LIN {X 0,Y 298.924,Z 413.247,A -85,B 0,C 180,E1 -16471.347,E2 -16471.347} C_VEL
LIN {X 0,Y 298.607,Z 413.287,A -85,B 0,C 180,E1 -16475.401,E2 -16475.401} C_VEL
LIN {X 0,Y 298.427,Z 413.313,A -85,B 0,C 180,E1 -16478.123,E2 -16478.123} C_VEL
LIN {X 0,Y 298.154,Z 413.46,A -85,B 0,C 180,E1 -16479.497,E2 -16479.497} C_VEL
LIN {X 0,Y 297.871,Z 417.389,A -85,B 0,C 180,E1 -16483.646,E2 -16483.646} C_VEL
LIN {X 0,Y 297.437,Z 421.454,A -85,B 0,C 180,E1 -16487.888,E2 -16487.888} C_VEL
LIN {X 0,Y 297.33,Z 423.309,A -85,B 0,C 180,E1 -16489.768,E2 -16489.768} C_VEL
LIN {X 0,Y 300.977,Z 438.073,A -85,B 0,C 180,E1 -16490.771,E2 -16490.771} C_VEL
LIN {X 0,Y 303.389,Z 449.477,A -85,B 0,C 180,E1 -16491.754,E2 -16491.754} C_VEL
LIN {X 0,Y 304.98,Z 459.069,A -85,B 0,C 180,E1 -16492.741,E2 -16492.741} C_VEL
LIN {X 0,Y 303.705,Z 471.172,A -85,B 0,C 180,E1 -16494.07,E2 -16494.07} C_VEL
LIN {X 0,Y 302.343,Z 482.034,A -85,B 0,C 180,E1 -16495.588,E2 -16495.588} C_VEL
LIN {X 0,Y 300.988,Z 492.034,A -85,B 0,C 180,E1 -16497.325,E2 -16497.325} C_VEL
LIN {X 0,Y 299.841,Z 500.268,A -85,B 0,C 180,E1 -16499.101,E2 -16499.101} C_VEL
LIN {X 0,Y 298.694,Z 508.025,A -85,B 0,C 180,E1 -16501.173,E2 -16501.173} C_VEL
LIN {X 0,Y 298.042,Z 513.11,A -85,B 0,C 180,E1 -16502.843,E2 -16502.843} C_VEL
LIN {X 0,Y 297.488,Z 517.392,A -85,B 0,C 180,E1 -16504.539,E2 -16504.539} C_VEL
LIN {X 0,Y 296.854,Z 522.403,A -85,B 0,C 180,E1 -16507.174,E2 -16507.174} C_VEL
LIN {X 0,Y 296.651,Z 524.39,A -85,B 0,C 180,E1 -16508.574,E2 -16508.574} C_VEL
LIN {X 0,Y 296.39,Z 526.457,A -85,B 0,C 180,E1 -16510.643,E2 -16510.643} C_VEL
LIN {X 0,Y 296.318,Z 527.731,A -85,B 0,C 180,E1 -16513.456,E2 -16513.456} C_VEL
LIN {X 0,Y 296.377,Z 527.652,A -85,B 0,C 180,E1 -16515.347,E2 -16515.347} C_VEL
LIN {X 0,Y 296.62,Z 526.789,A -85,B 0,C 180,E1 -16517.264,E2 -16517.264} C_VEL
LIN {X 0,Y 297.047,Z 525.061,A -85,B 0,C 180,E1 -16519.208,E2 -16519.208} C_VEL
LIN {X 0,Y 297.66,Z 522.432,A -85,B 0,C 180,E1 -16521.182,E2 -16521.182} C_VEL
LIN {X 0,Y 298.415,Z 518.77,A -85,B 0,C 180,E1 -16523.199,E2 -16523.199} C_VEL
LIN {X 0,Y 299.433,Z 513.955,A -85,B 0,C 180,E1 -16525.232,E2 -16525.232} C_VEL
LIN {X 0,Y 300.922,Z 507.021,A -85,B 0,C 180,E1 -16527.509,E2 -16527.509} C_VEL
LIN {X 0,Y 302.361,Z 500.069,A -85,B 0,C 180,E1 -16529.317,E2 -16529.317} C_VEL
LIN {X 0,Y 304.36,Z 490.374,A -85,B 0,C 180,E1 -16531.336,E2 -16531.336} C_VEL
LIN {X 0,Y 306.05,Z 481.363,A -85,B 0,C 180,E1 -16532.849,E2 -16532.849} C_VEL
LIN {X 0,Y 307.84,Z 470.675,A -85,B 0,C 180,E1 -16534.293,E2 -16534.293} C_VEL
LIN {X 0,Y 308.746,Z 463.633,A -85,B 0,C 180,E1 -16535.095,E2 -16535.095} C_VEL
LIN {X 0,Y 307.123,Z 453.705,A -85,B 0,C 180,E1 -16536.322,E2 -16536.322} C_VEL
LIN {X 0,Y 304.252,Z 442.437,A -85,B 0,C 180,E1 -16537.597,E2 -16537.597} C_VEL
LIN {X 0,Y 300.037,Z 430.605,A -85,B 0,C 180,E1 -16538.846,E2 -16538.846} C_VEL
LIN {X 0,Y 298.096,Z 425.478,A -85,B 0,C 180,E1 -16539.333,E2 -16539.333} C_VEL
LIN {X 0,Y 298.371,Z 422.974,A -85,B 0,C 180,E1 -16542.169,E2 -16542.169} C_VEL
LIN {X 0,Y 298.739,Z 420.721,A -85,B 0,C 180,E1 -16545.002,E2 -16545.002} C_VEL
LIN {X 0,Y 298.89,Z 419.097,A -85,B 0,C 180,E1 -16547.183,E2 -16547.183} C_VEL
LIN {X 0,Y 298.349,Z 418.395,A -85,B 0,C 180,E1 -16548.301,E2 -16548.301} C_VEL
LIN {X 0,Y 295.711,Z 417.616,A -85,B 0,C 180,E1 -16550.135,E2 -16550.135} C_VEL
LIN {X 0,Y 292.496,Z 416.764,A -85,B 0,C 180,E1 -16552.386,E2 -16552.386} C_VEL
LIN {X 0,Y 292.069,Z 416.37,A -85,B 0,C 180,E1 -16553.16,E2 -16553.16} C_VEL
LIN {X 0,Y 291.789,Z 414.141,A -85,B 0,C 180,E1 -16557.239,E2 -16557.239} C_VEL
LIN {X 0,Y 291.977,Z 414.116,A -85,B 0,C 180,E1 -16560,E2 -16560} C_VEL
LIN {X 0,Y 291.786,Z 414.138,A -85,B 0,C 180,E1 -16562.761,E2 -16562.761} C_VEL
LIN {X 0,Y 291.743,Z 414.145,A -85,B 0,C 180,E1 -16566.918,E2 -16566.918} C_VEL
LIN {X 0,Y 291.626,Z 414.16,A -85,B 0,C 180,E1 -16569.712,E2 -16569.712} C_VEL
LIN {X 0,Y 291.518,Z 414.174,A -85,B 0,C 180,E1 -16573.951,E2 -16573.951} C_VEL
LIN {X 0,Y 291.483,Z 414.178,A -85,B 0,C 180,E1 -16576.818,E2 -16576.818} C_VEL
LIN {X 0,Y 291.447,Z 414.181,A -85,B 0,C 180,E1 -16579.875,E2 -16579.875} C_VEL
LIN {X 0,Y 291.397,Z 414.184,A -85,B 0,C 180,E1 -16584.206,E2 -16584.206} C_VEL
LIN {X 0,Y 291.42,Z 414.185,A -85,B 0,C 180,E1 -16587.272,E2 -16587.272} C_VEL
LIN {X 0,Y 291.335,Z 414.196,A -85,B 0,C 180,E1 -16590.437,E2 -16590.437} C_VEL
LIN {X 0,Y 291.342,Z 414.197,A -85,B 0,C 180,E1 -16593.699,E2 -16593.699} C_VEL
LIN {X 0,Y 291.384,Z 414.193,A -85,B 0,C 180,E1 -16595.371,E2 -16595.371} C_VEL
LIN {X 0,Y 291.576,Z 415.192,A -85,B 0,C 180,E1 -16597.307,E2 -16597.307} C_VEL
LIN {X 0,Y 291.962,Z 417.466,A -85,B 0,C 180,E1 -16600.537,E2 -16600.537} C_VEL
LIN {X 0,Y 292.454,Z 420.429,A -85,B 0,C 180,E1 -16604.179,E2 -16604.179} C_VEL
LIN {X 0,Y 293.009,Z 423.998,A -85,B 0,C 180,E1 -16608.035,E2 -16608.035} C_VEL
LIN {X 0,Y 293.495,Z 427.586,A -85,B 0,C 180,E1 -16611.495,E2 -16611.495} C_VEL
LIN {X 0,Y 293.526,Z 431.017,A -85,B 0,C 180,E1 -16614.496,E2 -16614.496} C_VEL
LIN {X 0,Y 292.934,Z 434.304,A -85,B 0,C 180,E1 -16617.11,E2 -16617.11} C_VEL
LIN {X 0,Y 291.919,Z 439.75,A -85,B 0,C 180,E1 -16621.217,E2 -16621.217} C_VEL
LIN {X 0,Y 291.619,Z 441.928,A -85,B 0,C 180,E1 -16622.82,E2 -16622.82} C_VEL
LIN {X 0,Y 292.601,Z 445.427,A -85,B 0,C 180,E1 -16623.121,E2 -16623.121} C_VEL
LIN {X 0,Y 296.153,Z 457.869,A -85,B 0,C 180,E1 -16624.282,E2 -16624.282} C_VEL
LIN {X 0,Y 298.394,Z 469.519,A -85,B 0,C 180,E1 -16625.468,E2 -16625.468} C_VEL
LIN {X 0,Y 299.71,Z 481.807,A -85,B 0,C 180,E1 -16626.864,E2 -16626.864} C_VEL
LIN {X 0,Y 299.877,Z 491.89,A -85,B 0,C 180,E1 -16628.159,E2 -16628.159} C_VEL
LIN {X 0,Y 298.451,Z 500.372,A -85,B 0,C 180,E1 -16629.316,E2 -16629.316} C_VEL
LIN {X 0,Y 296.409,Z 510.463,A -85,B 0,C 180,E1 -16630.973,E2 -16630.973} C_VEL
LIN {X 0,Y 294.65,Z 519.181,A -85,B 0,C 180,E1 -16632.756,E2 -16632.756} C_VEL
LIN {X 0,Y 293.172,Z 526.933,A -85,B 0,C 180,E1 -16634.711,E2 -16634.711} C_VEL
LIN {X 0,Y 291.663,Z 533.586,A -85,B 0,C 180,E1 -16636.767,E2 -16636.767} C_VEL
LIN {X 0,Y 290.708,Z 538.932,A -85,B 0,C 180,E1 -16638.849,E2 -16638.849} C_VEL
LIN {X 0,Y 290.033,Z 543.121,A -85,B 0,C 180,E1 -16640.938,E2 -16640.938} C_VEL
LIN {X 0,Y 289.609,Z 546.265,A -85,B 0,C 180,E1 -16643.031,E2 -16643.031} C_VEL
LIN {X 0,Y 289.475,Z 547.919,A -85,B 0,C 180,E1 -16644.513,E2 -16644.513} C_VEL
LIN {X 0,Y 289.475,Z 549.701,A -85,B 0,C 180,E1 -16647.217,E2 -16647.217} C_VEL
LIN {X 0,Y 289.459,Z 550.041,A -85,B 0,C 180,E1 -16648.609,E2 -16648.609} C_VEL
LIN {X 0,Y 289.498,Z 549.984,A -85,B 0,C 180,E1 -16650.001,E2 -16650.001} C_VEL
LIN {X 0,Y 289.467,Z 549.479,A -85,B 0,C 180,E1 -16651.392,E2 -16651.392} C_VEL
LIN {X 0,Y 289.49,Z 548.572,A -85,B 0,C 180,E1 -16652.784,E2 -16652.784} C_VEL
LIN {X 0,Y 289.467,Z 547.256,A -85,B 0,C 180,E1 -16654.177,E2 -16654.177} C_VEL
LIN {X 0,Y 289.555,Z 544.436,A -85,B 0,C 180,E1 -16656.271,E2 -16656.271} C_VEL
LIN {X 0,Y 289.846,Z 540.562,A -85,B 0,C 180,E1 -16658.366,E2 -16658.366} C_VEL
LIN {X 0,Y 290.351,Z 535.532,A -85,B 0,C 180,E1 -16660.46,E2 -16660.46} C_VEL
LIN {X 0,Y 291.089,Z 529.192,A -85,B 0,C 180,E1 -16662.551,E2 -16662.551} C_VEL
LIN {X 0,Y 292.231,Z 521.244,A -85,B 0,C 180,E1 -16664.627,E2 -16664.627} C_VEL
LIN {X 0,Y 293.404,Z 513.15,A -85,B 0,C 180,E1 -16666.347,E2 -16666.347} C_VEL
LIN {X 0,Y 294.728,Z 503.29,A -85,B 0,C 180,E1 -16668.059,E2 -16668.059} C_VEL
LIN {X 0,Y 296.272,Z 492.31,A -85,B 0,C 180,E1 -16669.577,E2 -16669.577} C_VEL
LIN {X 0,Y 296.655,Z 488.023,A -85,B 0,C 180,E1 -16670.092,E2 -16670.092} C_VEL
LIN {X 0,Y 295.753,Z 476.605,A -85,B 0,C 180,E1 -16671.347,E2 -16671.347} C_VEL
LIN {X 0,Y 294.197,Z 463.998,A -85,B 0,C 180,E1 -16672.472,E2 -16672.472} C_VEL
LIN {X 0,Y 292.088,Z 451.05,A -85,B 0,C 180,E1 -16673.378,E2 -16673.378} C_VEL
LIN {X 0,Y 290.748,Z 443.879,A -85,B 0,C 180,E1 -16673.794,E2 -16673.794} C_VEL
LIN {X 0,Y 291.476,Z 437.644,A -85,B 0,C 180,E1 -16678.046,E2 -16678.046} C_VEL
LIN {X 0,Y 292.238,Z 432.07,A -85,B 0,C 180,E1 -16681.943,E2 -16681.943} C_VEL
LIN {X 0,Y 292.974,Z 427.301,A -85,B 0,C 180,E1 -16685.352,E2 -16685.352} C_VEL
LIN {X 0,Y 292.931,Z 423.009,A -85,B 0,C 180,E1 -16688.594,E2 -16688.594} C_VEL
LIN {X 0,Y 292.132,Z 418.347,A -85,B 0,C 180,E1 -16692.347,E2 -16692.347} C_VEL
LIN {X 0,Y 291.364,Z 414.193,A -85,B 0,C 180,E1 -16696.046,E2 -16696.046} C_VEL
LIN {X 0,Y 291.38,Z 414.189,A -85,B 0,C 180,E1 -16700.519,E2 -16700.519} C_VEL
LIN {X 0,Y 291.406,Z 414.186,A -85,B 0,C 180,E1 -16702.919,E2 -16702.919} C_VEL
LIN {X 0,Y 291.346,Z 414.191,A -85,B 0,C 180,E1 -16706.302,E2 -16706.302} C_VEL
LIN {X 0,Y 291.389,Z 414.185,A -85,B 0,C 180,E1 -16710.26,E2 -16710.26} C_VEL
LIN {X 0,Y 291.414,Z 414.18,A -85,B 0,C 180,E1 -16714.271,E2 -16714.271} C_VEL
LIN {X 0,Y 291.383,Z 414.19,A -85,B 0,C 180,E1 -16717.299,E2 -16717.299} C_VEL
LIN {X 0,Y 291.459,Z 414.177,A -85,B 0,C 180,E1 -16720.27,E2 -16720.27} C_VEL
LIN {X 0,Y 291.557,Z 414.166,A -85,B 0,C 180,E1 -16724.624,E2 -16724.624} C_VEL
LIN {X 0,Y 291.538,Z 414.17,A -85,B 0,C 180,E1 -16728.881,E2 -16728.881} C_VEL
LIN {X 0,Y 291.71,Z 414.146,A -85,B 0,C 180,E1 -16731.688,E2 -16731.688} C_VEL
LIN {X 0,Y 291.631,Z 414.156,A -85,B 0,C 180,E1 -16734.468,E2 -16734.468} C_VEL
LIN {X 0,Y 291.889,Z 414.125,A -85,B 0,C 180,E1 -16738.62,E2 -16738.62} C_VEL
LIN {X 0,Y 291.89,Z 414.124,A -85,B 0,C 180,E1 -16741.38,E2 -16741.38} C_VEL
LIN {X 0,Y 291.747,Z 414.145,A -85,B 0,C 180,E1 -16746.918,E2 -16746.918} C_VEL
LIN {X 0,Y 291.631,Z 414.155,A -85,B 0,C 180,E1 -16749.712,E2 -16749.712} C_VEL
LIN {X 0,Y 291.523,Z 414.166,A -85,B 0,C 180,E1 -16753.95,E2 -16753.95} C_VEL
LIN {X 0,Y 291.488,Z 414.171,A -85,B 0,C 180,E1 -16756.818,E2 -16756.818} C_VEL
LIN {X 0,Y 291.452,Z 414.173,A -85,B 0,C 180,E1 -16759.875,E2 -16759.875} C_VEL
LIN {X 0,Y 291.402,Z 414.184,A -85,B 0,C 180,E1 -16764.205,E2 -16764.205} C_VEL
LIN {X 0,Y 291.427,Z 414.182,A -85,B 0,C 180,E1 -16767.271,E2 -16767.271} C_VEL
LIN {X 0,Y 291.338,Z 414.194,A -85,B 0,C 180,E1 -16770.437,E2 -16770.437} C_VEL
LIN {X 0,Y 291.346,Z 414.187,A -85,B 0,C 180,E1 -16773.698,E2 -16773.698} C_VEL
LIN {X 0,Y 291.377,Z 414.184,A -85,B 0,C 180,E1 -16777.254,E2 -16777.254} C_VEL
LIN {X 0,Y 291.334,Z 414.196,A -85,B 0,C 180,E1 -16780.642,E2 -16780.642} C_VEL
LIN {X 0,Y 291.291,Z 414.201,A -85,B 0,C 180,E1 -16784.402,E2 -16784.402} C_VEL
LIN {X 0,Y 291.328,Z 414.195,A -85,B 0,C 180,E1 -16788.404,E2 -16788.404} C_VEL
LIN {X 0,Y 291.366,Z 414.185,A -85,B 0,C 180,E1 -16791.16,E2 -16791.16} C_VEL
LIN {X 0,Y 291.387,Z 414.19,A -85,B 0,C 180,E1 -16794.629,E2 -16794.629} C_VEL
LIN {X 0,Y 291.372,Z 414.189,A -85,B 0,C 180,E1 -16797.95,E2 -16797.95} C_VEL
LIN {X 0,Y 291.378,Z 414.186,A -85,B 0,C 180,E1 -16801.158,E2 -16801.158} C_VEL
LIN {X 0,Y 291.414,Z 414.183,A -85,B 0,C 180,E1 -16804.271,E2 -16804.271} C_VEL
LIN {X 0,Y 291.391,Z 414.186,A -85,B 0,C 180,E1 -16807.3,E2 -16807.3} C_VEL
LIN {X 0,Y 291.46,Z 414.18,A -85,B 0,C 180,E1 -16810.27,E2 -16810.27} C_VEL
LIN {X 0,Y 291.557,Z 414.168,A -85,B 0,C 180,E1 -16814.623,E2 -16814.623} C_VEL
LIN {X 0,Y 291.539,Z 414.167,A -85,B 0,C 180,E1 -16818.88,E2 -16818.88} C_VEL
LIN {X 0,Y 291.712,Z 414.146,A -85,B 0,C 180,E1 -16821.688,E2 -16821.688} C_VEL
LIN {X 0,Y 291.632,Z 414.157,A -85,B 0,C 180,E1 -16824.468,E2 -16824.468} C_VEL
LIN {X 0,Y 291.89,Z 414.126,A -85,B 0,C 180,E1 -16828.62,E2 -16828.62} C_VEL
LIN {X 0,Y 291.89,Z 414.124,A -85,B 0,C 180,E1 -16831.379,E2 -16831.379} C_VEL
LIN {X 0,Y 291.568,Z 414.165,A -85,B 0,C 180,E1 -16835.532,E2 -16835.532} C_VEL
LIN {X 0,Y 291.318,Z 414.198,A -85,B 0,C 180,E1 -16838.46,E2 -16838.46} C_VEL
LIN {X 0,Y 291.074,Z 414.562,A -85,B 0,C 180,E1 -16839.73,E2 -16839.73} C_VEL
LIN {X 0,Y 290.787,Z 418.522,A -85,B 0,C 180,E1 -16843.986,E2 -16843.986} C_VEL
LIN {X 0,Y 290.341,Z 422.658,A -85,B 0,C 180,E1 -16848.341,E2 -16848.341} C_VEL
LIN {X 0,Y 290.311,Z 423.576,A -85,B 0,C 180,E1 -16849.299,E2 -16849.299} C_VEL
LIN {X 0,Y 293.844,Z 437.855,A -85,B 0,C 180,E1 -16850.291,E2 -16850.291} C_VEL
LIN {X 0,Y 296.457,Z 450.147,A -85,B 0,C 180,E1 -16851.375,E2 -16851.375} C_VEL
LIN {X 0,Y 298.112,Z 460.988,A -85,B 0,C 180,E1 -16852.525,E2 -16852.525} C_VEL
LIN {X 0,Y 296.663,Z 473.085,A -85,B 0,C 180,E1 -16853.934,E2 -16853.934} C_VEL
LIN {X 0,Y 295.246,Z 484.104,A -85,B 0,C 180,E1 -16855.559,E2 -16855.559} C_VEL
LIN {X 0,Y 293.834,Z 493.735,A -85,B 0,C 180,E1 -16857.342,E2 -16857.342} C_VEL
LIN {X 0,Y 292.58,Z 502.458,A -85,B 0,C 180,E1 -16859.347,E2 -16859.347} C_VEL
LIN {X 0,Y 291.586,Z 509.032,A -85,B 0,C 180,E1 -16861.211,E2 -16861.211} C_VEL
LIN {X 0,Y 290.871,Z 514.22,A -85,B 0,C 180,E1 -16863.012,E2 -16863.012} C_VEL
LIN {X 0,Y 290.115,Z 519.959,A -85,B 0,C 180,E1 -16865.548,E2 -16865.548} C_VEL
LIN {X 0,Y 289.613,Z 524.142,A -85,B 0,C 180,E1 -16868.169,E2 -16868.169} C_VEL
LIN {X 0,Y 289.292,Z 526.943,A -85,B 0,C 180,E1 -16870.989,E2 -16870.989} C_VEL
LIN {X 0,Y 289.227,Z 527.954,A -85,B 0,C 180,E1 -16873.199,E2 -16873.199} C_VEL
LIN {X 0,Y 289.272,Z 528.012,A -85,B 0,C 180,E1 -16875.205,E2 -16875.205} C_VEL
LIN {X 0,Y 289.51,Z 527.234,A -85,B 0,C 180,E1 -16877.179,E2 -16877.179} C_VEL
LIN {X 0,Y 289.932,Z 525.691,A -85,B 0,C 180,E1 -16879.119,E2 -16879.119} C_VEL
LIN {X 0,Y 290.531,Z 523.396,A -85,B 0,C 180,E1 -16881.028,E2 -16881.028} C_VEL
LIN {X 0,Y 291.202,Z 520.364,A -85,B 0,C 180,E1 -16882.889,E2 -16882.889} C_VEL
LIN {X 0,Y 292.379,Z 515.096,A -85,B 0,C 180,E1 -16885.295,E2 -16885.295} C_VEL
LIN {X 0,Y 293.919,Z 508.359,A -85,B 0,C 180,E1 -16887.643,E2 -16887.643} C_VEL
LIN {X 0,Y 295.487,Z 501.391,A -85,B 0,C 180,E1 -16889.563,E2 -16889.563} C_VEL
LIN {X 0,Y 297.407,Z 492.754,A -85,B 0,C 180,E1 -16891.468,E2 -16891.468} C_VEL
LIN {X 0,Y 299.46,Z 482.345,A -85,B 0,C 180,E1 -16893.305,E2 -16893.305} C_VEL
LIN {X 0,Y 301.37,Z 471.589,A -85,B 0,C 180,E1 -16894.813,E2 -16894.813} C_VEL
LIN {X 0,Y 302.242,Z 466.062,A -85,B 0,C 180,E1 -16895.459,E2 -16895.459} C_VEL
LIN {X 0,Y 301.069,Z 457.199,A -85,B 0,C 180,E1 -16896.619,E2 -16896.619} C_VEL
LIN {X 0,Y 298.662,Z 446.906,A -85,B 0,C 180,E1 -16897.883,E2 -16897.883} C_VEL
LIN {X 0,Y 294.909,Z 435.322,A -85,B 0,C 180,E1 -16899.193,E2 -16899.193} C_VEL
LIN {X 0,Y 291.251,Z 426.22,A -85,B 0,C 180,E1 -16900.173,E2 -16900.173} C_VEL
LIN {X 0,Y 291.162,Z 425.602,A -85,B 0,C 180,E1 -16900.249,E2 -16900.249} C_VEL
LIN {X 0,Y 291.656,Z 422.178,A -85,B 0,C 180,E1 -16904.629,E2 -16904.629} C_VEL
LIN {X 0,Y 291.921,Z 420.084,A -85,B 0,C 180,E1 -16907.486,E2 -16907.486} C_VEL
LIN {X 0,Y 292.135,Z 418.019,A -85,B 0,C 180,E1 -16910.517,E2 -16910.517} C_VEL
LIN {X 0,Y 292.069,Z 416.37,A -85,B 0,C 180,E1 -16913.16,E2 -16913.16} C_VEL
LIN {X 0,Y 291.228,Z 415.855,A -85,B 0,C 180,E1 -16914.304,E2 -16914.304} C_VEL
LIN {X 0,Y 288.277,Z 415.39,A -85,B 0,C 180,E1 -16916.174,E2 -16916.174} C_VEL
LIN {X 0,Y 285.901,Z 415.125,A -85,B 0,C 180,E1 -16917.695,E2 -16917.695} C_VEL
LIN {X 0,Y 284.93,Z 415.01,A -85,B 0,C 180,E1 -16918.873,E2 -16918.873} C_VEL
LIN {X 0,Y 284.871,Z 414.999,A -85,B 0,C 180,E1 -16919.272,E2 -16919.272} C_VEL
LIN {X 0,Y 284.741,Z 415.016,A -85,B 0,C 180,E1 -16922.83,E2 -16922.83} C_VEL
LIN {X 0,Y 284.695,Z 415.023,A -85,B 0,C 180,E1 -16927.09,E2 -16927.09} C_VEL
LIN {X 0,Y 284.563,Z 415.04,A -85,B 0,C 180,E1 -16929.956,E2 -16929.956} C_VEL
LIN {X 0,Y 284.478,Z 415.05,A -85,B 0,C 180,E1 -16934.303,E2 -16934.303} C_VEL
LIN {X 0,Y 284.422,Z 415.057,A -85,B 0,C 180,E1 -16937.249,E2 -16937.249} C_VEL
LIN {X 0,Y 284.375,Z 415.063,A -85,B 0,C 180,E1 -16940.243,E2 -16940.243} C_VEL
LIN {X 0,Y 284.366,Z 415.06,A -85,B 0,C 180,E1 -16943.876,E2 -16943.876} C_VEL
LIN {X 0,Y 284.394,Z 415.06,A -85,B 0,C 180,E1 -16947.174,E2 -16947.174} C_VEL
LIN {X 0,Y 284.293,Z 415.074,A -85,B 0,C 180,E1 -16951.275,E2 -16951.275} C_VEL
LIN {X 0,Y 284.343,Z 415.233,A -85,B 0,C 180,E1 -16954.645,E2 -16954.645} C_VEL
LIN {X 0,Y 284.716,Z 417.331,A -85,B 0,C 180,E1 -16958.105,E2 -16958.105} C_VEL
LIN {X 0,Y 285.185,Z 419.912,A -85,B 0,C 180,E1 -16961.712,E2 -16961.712} C_VEL
LIN {X 0,Y 285.665,Z 423.069,A -85,B 0,C 180,E1 -16965.518,E2 -16965.518} C_VEL
LIN {X 0,Y 286.294,Z 426.86,A -85,B 0,C 180,E1 -16969.552,E2 -16969.552} C_VEL
LIN {X 0,Y 286.584,Z 429.606,A -85,B 0,C 180,E1 -16972.188,E2 -16972.188} C_VEL
LIN {X 0,Y 286.553,Z 431.679,A -85,B 0,C 180,E1 -16974.034,E2 -16974.034} C_VEL
LIN {X 0,Y 285.833,Z 435.598,A -85,B 0,C 180,E1 -16977.254,E2 -16977.254} C_VEL
LIN {X 0,Y 284.724,Z 441.631,A -85,B 0,C 180,E1 -16981.907,E2 -16981.907} C_VEL
LIN {X 0,Y 285.569,Z 444.764,A -85,B 0,C 180,E1 -16982.169,E2 -16982.169} C_VEL
LIN {X 0,Y 288.858,Z 455.345,A -85,B 0,C 180,E1 -16983.231,E2 -16983.231} C_VEL
LIN {X 0,Y 291.371,Z 466.632,A -85,B 0,C 180,E1 -16984.421,E2 -16984.421} C_VEL
LIN {X 0,Y 292.858,Z 478.362,A -85,B 0,C 180,E1 -16985.773,E2 -16985.773} C_VEL
LIN {X 0,Y 293.353,Z 489.212,A -85,B 0,C 180,E1 -16987.184,E2 -16987.184} C_VEL
LIN {X 0,Y 293.064,Z 494.991,A -85,B 0,C 180,E1 -16987.995,E2 -16987.995} C_VEL
LIN {X 0,Y 290.931,Z 505.092,A -85,B 0,C 180,E1 -16989.497,E2 -16989.497} C_VEL
LIN {X 0,Y 288.953,Z 514.258,A -85,B 0,C 180,E1 -16991.2,E2 -16991.2} C_VEL
LIN {X 0,Y 287.079,Z 523.236,A -85,B 0,C 180,E1 -16993.283,E2 -16993.283} C_VEL
LIN {X 0,Y 285.534,Z 530.531,A -85,B 0,C 180,E1 -16995.388,E2 -16995.388} C_VEL
LIN {X 0,Y 284.305,Z 535.504,A -85,B 0,C 180,E1 -16997.146,E2 -16997.146} C_VEL
LIN {X 0,Y 283.449,Z 540.371,A -85,B 0,C 180,E1 -16999.284,E2 -16999.284} C_VEL
LIN {X 0,Y 282.807,Z 544.146,A -85,B 0,C 180,E1 -17001.426,E2 -17001.426} C_VEL
LIN {X 0,Y 282.556,Z 546.12,A -85,B 0,C 180,E1 -17002.857,E2 -17002.857} C_VEL
LIN {X 0,Y 282.371,Z 547.92,A -85,B 0,C 180,E1 -17004.608,E2 -17004.608} C_VEL
LIN {X 0,Y 282.379,Z 549.461,A -85,B 0,C 180,E1 -17007.147,E2 -17007.147} C_VEL
LIN {X 0,Y 282.38,Z 549.778,A -85,B 0,C 180,E1 -17008.574,E2 -17008.574} C_VEL
LIN {X 0,Y 282.415,Z 549.677,A -85,B 0,C 180,E1 -17010.001,E2 -17010.001} C_VEL
LIN {X 0,Y 282.388,Z 549.141,A -85,B 0,C 180,E1 -17011.427,E2 -17011.427} C_VEL
LIN {X 0,Y 282.417,Z 548.209,A -85,B 0,C 180,E1 -17012.853,E2 -17012.853} C_VEL
LIN {X 0,Y 282.409,Z 545.407,A -85,B 0,C 180,E1 -17015.474,E2 -17015.474} C_VEL
LIN {X 0,Y 282.672,Z 541.5,A -85,B 0,C 180,E1 -17017.86,E2 -17017.86} C_VEL
LIN {X 0,Y 283.128,Z 536.8,A -85,B 0,C 180,E1 -17020.007,E2 -17020.007} C_VEL
LIN {X 0,Y 283.944,Z 529.697,A -85,B 0,C 180,E1 -17022.508,E2 -17022.508} C_VEL
LIN {X 0,Y 285.128,Z 521.998,A -85,B 0,C 180,E1 -17024.635,E2 -17024.635} C_VEL
LIN {X 0,Y 286.385,Z 513.316,A -85,B 0,C 180,E1 -17026.554,E2 -17026.554} C_VEL
LIN {X 0,Y 287.774,Z 503.414,A -85,B 0,C 180,E1 -17028.327,E2 -17028.327} C_VEL
LIN {X 0,Y 289.357,Z 492.563,A -85,B 0,C 180,E1 -17029.88,E2 -17029.88} C_VEL
LIN {X 0,Y 289.697,Z 488.295,A -85,B 0,C 180,E1 -17030.41,E2 -17030.41} C_VEL
LIN {X 0,Y 288.705,Z 476.025,A -85,B 0,C 180,E1 -17031.797,E2 -17031.797} C_VEL
LIN {X 0,Y 287.077,Z 463.033,A -85,B 0,C 180,E1 -17032.983,E2 -17032.983} C_VEL
LIN {X 0,Y 284.861,Z 449.796,A -85,B 0,C 180,E1 -17033.92,E2 -17033.92} C_VEL
LIN {X 0,Y 283.728,Z 443.632,A -85,B 0,C 180,E1 -17034.283,E2 -17034.283} C_VEL
LIN {X 0,Y 284.56,Z 437.226,A -85,B 0,C 180,E1 -17038.791,E2 -17038.791} C_VEL
LIN {X 0,Y 285.403,Z 431.635,A -85,B 0,C 180,E1 -17042.803,E2 -17042.803} C_VEL
LIN {X 0,Y 285.979,Z 427.584,A -85,B 0,C 180,E1 -17045.807,E2 -17045.807} C_VEL
LIN {X 0,Y 285.853,Z 423.634,A -85,B 0,C 180,E1 -17048.872,E2 -17048.872} C_VEL
LIN {X 0,Y 285.143,Z 419.473,A -85,B 0,C 180,E1 -17052.318,E2 -17052.318} C_VEL
LIN {X 0,Y 284.306,Z 415.072,A -85,B 0,C 180,E1 -17056.199,E2 -17056.199} C_VEL
LIN {X 0,Y 284.308,Z 415.07,A -85,B 0,C 180,E1 -17060.024,E2 -17060.024} C_VEL
LIN {X 0,Y 284.332,Z 415.064,A -85,B 0,C 180,E1 -17063.614,E2 -17063.614} C_VEL
LIN {X 0,Y 284.309,Z 415.073,A -85,B 0,C 180,E1 -17067.19,E2 -17067.19} C_VEL
LIN {X 0,Y 284.36,Z 415.061,A -85,B 0,C 180,E1 -17070.376,E2 -17070.376} C_VEL
LIN {X 0,Y 284.376,Z 415.058,A -85,B 0,C 180,E1 -17073.586,E2 -17073.586} C_VEL
LIN {X 0,Y 284.368,Z 415.061,A -85,B 0,C 180,E1 -17076.707,E2 -17076.707} C_VEL
LIN {X 0,Y 284.405,Z 415.058,A -85,B 0,C 180,E1 -17081.262,E2 -17081.262} C_VEL
LIN {X 0,Y 284.494,Z 415.045,A -85,B 0,C 180,E1 -17084.459,E2 -17084.459} C_VEL
LIN {X 0,Y 284.49,Z 415.045,A -85,B 0,C 180,E1 -17088.601,E2 -17088.601} C_VEL
LIN {X 0,Y 284.66,Z 415.025,A -85,B 0,C 180,E1 -17091.481,E2 -17091.481} C_VEL
LIN {X 0,Y 284.602,Z 415.031,A -85,B 0,C 180,E1 -17094.331,E2 -17094.331} C_VEL
LIN {X 0,Y 284.855,Z 415,A -85,B 0,C 180,E1 -17098.586,E2 -17098.586} C_VEL
LIN {X 0,Y 284.856,Z 415,A -85,B 0,C 180,E1 -17101.414,E2 -17101.414} C_VEL
LIN {X 0,Y 284.699,Z 415.022,A -85,B 0,C 180,E1 -17107.09,E2 -17107.09} C_VEL
LIN {X 0,Y 284.568,Z 415.035,A -85,B 0,C 180,E1 -17109.955,E2 -17109.955} C_VEL
LIN {X 0,Y 284.483,Z 415.044,A -85,B 0,C 180,E1 -17114.303,E2 -17114.303} C_VEL
LIN {X 0,Y 284.427,Z 415.046,A -85,B 0,C 180,E1 -17117.248,E2 -17117.248} C_VEL
LIN {X 0,Y 284.38,Z 415.054,A -85,B 0,C 180,E1 -17120.242,E2 -17120.242} C_VEL
LIN {X 0,Y 284.37,Z 415.059,A -85,B 0,C 180,E1 -17123.875,E2 -17123.875} C_VEL
LIN {X 0,Y 284.401,Z 415.058,A -85,B 0,C 180,E1 -17127.174,E2 -17127.174} C_VEL
LIN {X 0,Y 284.297,Z 415.068,A -85,B 0,C 180,E1 -17131.274,E2 -17131.274} C_VEL
LIN {X 0,Y 284.342,Z 415.056,A -85,B 0,C 180,E1 -17135.348,E2 -17135.348} C_VEL
LIN {X 0,Y 284.313,Z 415.064,A -85,B 0,C 180,E1 -17138.169,E2 -17138.169} C_VEL
LIN {X 0,Y 284.27,Z 415.073,A -85,B 0,C 180,E1 -17142.124,E2 -17142.124} C_VEL
LIN {X 0,Y 284.256,Z 415.075,A -85,B 0,C 180,E1 -17146.189,E2 -17146.189} C_VEL
LIN {X 0,Y 284.308,Z 415.065,A -85,B 0,C 180,E1 -17150.024,E2 -17150.024} C_VEL
LIN {X 0,Y 284.352,Z 415.06,A -85,B 0,C 180,E1 -17153.617,E2 -17153.617} C_VEL
LIN {X 0,Y 284.309,Z 415.068,A -85,B 0,C 180,E1 -17157.189,E2 -17157.189} C_VEL
LIN {X 0,Y 284.357,Z 415.065,A -85,B 0,C 180,E1 -17160.375,E2 -17160.375} C_VEL
LIN {X 0,Y 284.376,Z 415.056,A -85,B 0,C 180,E1 -17163.586,E2 -17163.586} C_VEL
LIN {X 0,Y 284.371,Z 415.063,A -85,B 0,C 180,E1 -17166.707,E2 -17166.707} C_VEL
LIN {X 0,Y 284.405,Z 415.054,A -85,B 0,C 180,E1 -17171.261,E2 -17171.261} C_VEL
LIN {X 0,Y 284.494,Z 415.05,A -85,B 0,C 180,E1 -17174.459,E2 -17174.459} C_VEL
LIN {X 0,Y 284.49,Z 415.047,A -85,B 0,C 180,E1 -17178.601,E2 -17178.601} C_VEL
LIN {X 0,Y 284.662,Z 415.024,A -85,B 0,C 180,E1 -17181.481,E2 -17181.481} C_VEL
LIN {X 0,Y 284.603,Z 415.033,A -85,B 0,C 180,E1 -17184.331,E2 -17184.331} C_VEL
LIN {X 0,Y 284.856,Z 415.003,A -85,B 0,C 180,E1 -17188.586,E2 -17188.586} C_VEL
LIN {X 0,Y 284.856,Z 415,A -85,B 0,C 180,E1 -17191.413,E2 -17191.413} C_VEL
LIN {X 0,Y 284.528,Z 415.042,A -85,B 0,C 180,E1 -17195.67,E2 -17195.67} C_VEL
LIN {X 0,Y 284.265,Z 415.076,A -85,B 0,C 180,E1 -17198.53,E2 -17198.53} C_VEL
LIN {X 0,Y 284.048,Z 415.357,A -85,B 0,C 180,E1 -17199.613,E2 -17199.613} C_VEL
LIN {X 0,Y 283.771,Z 418.293,A -85,B 0,C 180,E1 -17202.879,E2 -17202.879} C_VEL
LIN {X 0,Y 283.493,Z 421.046,A -85,B 0,C 180,E1 -17205.824,E2 -17205.824} C_VEL
LIN {X 0,Y 283.282,Z 423.967,A -85,B 0,C 180,E1 -17208.815,E2 -17208.815} C_VEL
LIN {X 0,Y 286.608,Z 437.123,A -85,B 0,C 180,E1 -17209.746,E2 -17209.746} C_VEL
LIN {X 0,Y 289.204,Z 449.093,A -85,B 0,C 180,E1 -17210.818,E2 -17210.818} C_VEL
LIN {X 0,Y 291.146,Z 460.447,A -85,B 0,C 180,E1 -17212.045,E2 -17212.045} C_VEL
LIN {X 0,Y 290.64,Z 466.848,A -85,B 0,C 180,E1 -17212.761,E2 -17212.761} C_VEL
LIN {X 0,Y 289.262,Z 477.904,A -85,B 0,C 180,E1 -17214.227,E2 -17214.227} C_VEL
LIN {X 0,Y 287.908,Z 487.208,A -85,B 0,C 180,E1 -17215.744,E2 -17215.744} C_VEL
LIN {X 0,Y 286.704,Z 495.369,A -85,B 0,C 180,E1 -17217.362,E2 -17217.362} C_VEL
LIN {X 0,Y 285.355,Z 504.186,A -85,B 0,C 180,E1 -17219.509,E2 -17219.509} C_VEL
LIN {X 0,Y 284.348,Z 511.022,A -85,B 0,C 180,E1 -17221.605,E2 -17221.605} C_VEL
LIN {X 0,Y 283.474,Z 516.972,A -85,B 0,C 180,E1 -17223.905,E2 -17223.905} C_VEL
LIN {X 0,Y 282.996,Z 520.734,A -85,B 0,C 180,E1 -17225.756,E2 -17225.756} C_VEL
LIN {X 0,Y 282.479,Z 524.808,A -85,B 0,C 180,E1 -17228.461,E2 -17228.461} C_VEL
LIN {X 0,Y 282.244,Z 526.685,A -85,B 0,C 180,E1 -17230.346,E2 -17230.346} C_VEL
LIN {X 0,Y 282.139,Z 527.883,A -85,B 0,C 180,E1 -17232.264,E2 -17232.264} C_VEL
LIN {X 0,Y 282.126,Z 528.367,A -85,B 0,C 180,E1 -17234.226,E2 -17234.226} C_VEL
LIN {X 0,Y 282.283,Z 528.051,A -85,B 0,C 180,E1 -17236.22,E2 -17236.22} C_VEL
LIN {X 0,Y 282.633,Z 526.95,A -85,B 0,C 180,E1 -17238.243,E2 -17238.243} C_VEL
LIN {X 0,Y 283.174,Z 525.004,A -85,B 0,C 180,E1 -17240.297,E2 -17240.297} C_VEL
LIN {X 0,Y 284.176,Z 521.06,A -85,B 0,C 180,E1 -17243.011,E2 -17243.011} C_VEL
LIN {X 0,Y 285.428,Z 515.915,A -85,B 0,C 180,E1 -17245.506,E2 -17245.506} C_VEL
LIN {X 0,Y 286.908,Z 509.821,A -85,B 0,C 180,E1 -17247.741,E2 -17247.741} C_VEL
LIN {X 0,Y 288.439,Z 503.393,A -85,B 0,C 180,E1 -17249.63,E2 -17249.63} C_VEL
LIN {X 0,Y 290.464,Z 494.843,A -85,B 0,C 180,E1 -17251.651,E2 -17251.651} C_VEL
LIN {X 0,Y 292.341,Z 486.212,A -85,B 0,C 180,E1 -17253.302,E2 -17253.302} C_VEL
LIN {X 0,Y 294.276,Z 476.252,A -85,B 0,C 180,E1 -17254.853,E2 -17254.853} C_VEL
LIN {X 0,Y 295.801,Z 467.169,A -85,B 0,C 180,E1 -17256.013,E2 -17256.013} C_VEL
LIN {X 0,Y 294.466,Z 457.672,A -85,B 0,C 180,E1 -17257.324,E2 -17257.324} C_VEL
LIN {X 0,Y 291.968,Z 447.356,A -85,B 0,C 180,E1 -17258.649,E2 -17258.649} C_VEL
LIN {X 0,Y 287.89,Z 435.363,A -85,B 0,C 180,E1 -17260.104,E2 -17260.104} C_VEL
LIN {X 0,Y 285.055,Z 428.698,A -85,B 0,C 180,E1 -17260.893,E2 -17260.893} C_VEL
LIN {X 0,Y 284.223,Z 425.951,A -85,B 0,C 180,E1 -17261.186,E2 -17261.186} C_VEL
LIN {X 0,Y 284.741,Z 422.568,A -85,B 0,C 180,E1 -17265.711,E2 -17265.711} C_VEL
LIN {X 0,Y 284.995,Z 420.554,A -85,B 0,C 180,E1 -17268.622,E2 -17268.622} C_VEL
LIN {X 0,Y 285.183,Z 418.685,A -85,B 0,C 180,E1 -17271.497,E2 -17271.497} C_VEL
LIN {X 0,Y 284.932,Z 417.06,A -85,B 0,C 180,E1 -17274.338,E2 -17274.338} C_VEL
LIN {X 0,Y 284.854,Z 415.004,A -85,B 0,C 180,E1 -17278.586,E2 -17278.586} C_VEL
LIN {X 0,Y 284.871,Z 414.999,A -85,B 0,C 180,E1 -17279.272,E2 -17279.272} C_VEL
LIN {X 0,Y 284.201,Z 415.084,A -85,B 0,C 180,E1 -17280.451,E2 -17280.451} C_VEL
LIN {X 0,Y 281.167,Z 415.46,A -85,B 0,C 180,E1 -17282.365,E2 -17282.365} C_VEL
LIN {X 0,Y 278.612,Z 415.781,A -85,B 0,C 180,E1 -17283.922,E2 -17283.922} C_VEL
LIN {X 0,Y 277.582,Z 415.91,A -85,B 0,C 180,E1 -17285.133,E2 -17285.133} C_VEL
LIN {X 0,Y 277.535,Z 415.914,A -85,B 0,C 180,E1 -17285.543,E2 -17285.543} C_VEL
LIN {X 0,Y 277.612,Z 415.906,A -85,B 0,C 180,E1 -17288.737,E2 -17288.737} C_VEL
LIN {X 0,Y 277.413,Z 415.93,A -85,B 0,C 180,E1 -17293.18,E2 -17293.18} C_VEL
LIN {X 0,Y 277.403,Z 415.931,A -85,B 0,C 180,E1 -17296.182,E2 -17296.182} C_VEL
LIN {X 0,Y 277.342,Z 415.939,A -85,B 0,C 180,E1 -17300.35,E2 -17300.35} C_VEL
LIN {X 0,Y 277.316,Z 415.937,A -85,B 0,C 180,E1 -17304.171,E2 -17304.171} C_VEL
LIN {X 0,Y 277.323,Z 415.942,A -85,B 0,C 180,E1 -17307.506,E2 -17307.506} C_VEL
LIN {X 0,Y 277.269,Z 415.948,A -85,B 0,C 180,E1 -17310.482,E2 -17310.482} C_VEL
LIN {X 0,Y 277.287,Z 416.154,A -85,B 0,C 180,E1 -17313.239,E2 -17313.239} C_VEL
LIN {X 0,Y 277.572,Z 417.557,A -85,B 0,C 180,E1 -17315.884,E2 -17315.884} C_VEL
LIN {X 0,Y 277.919,Z 419.664,A -85,B 0,C 180,E1 -17319.213,E2 -17319.213} C_VEL
LIN {X 0,Y 278.406,Z 422.406,A -85,B 0,C 180,E1 -17322.968,E2 -17322.968} C_VEL
LIN {X 0,Y 278.966,Z 425.936,A -85,B 0,C 180,E1 -17327.141,E2 -17327.141} C_VEL
LIN {X 0,Y 279.263,Z 427.793,A -85,B 0,C 180,E1 -17329.133,E2 -17329.133} C_VEL
LIN {X 0,Y 279.49,Z 429.864,A -85,B 0,C 180,E1 -17331.217,E2 -17331.217} C_VEL
LIN {X 0,Y 279.559,Z 432.373,A -85,B 0,C 180,E1 -17333.559,E2 -17333.559} C_VEL
LIN {X 0,Y 279.037,Z 435.603,A -85,B 0,C 180,E1 -17336.352,E2 -17336.352} C_VEL
LIN {X 0,Y 277.886,Z 441.268,A -85,B 0,C 180,E1 -17340.905,E2 -17340.905} C_VEL
LIN {X 0,Y 279,Z 444.991,A -85,B 0,C 180,E1 -17341.265,E2 -17341.265} C_VEL
LIN {X 0,Y 282.489,Z 456.404,A -85,B 0,C 180,E1 -17342.478,E2 -17342.478} C_VEL
LIN {X 0,Y 284.965,Z 467.644,A -85,B 0,C 180,E1 -17343.755,E2 -17343.755} C_VEL
LIN {X 0,Y 286.423,Z 479.622,A -85,B 0,C 180,E1 -17345.214,E2 -17345.214} C_VEL
LIN {X 0,Y 286.831,Z 490.082,A -85,B 0,C 180,E1 -17346.641,E2 -17346.641} C_VEL
LIN {X 0,Y 286.289,Z 496.878,A -85,B 0,C 180,E1 -17347.636,E2 -17347.636} C_VEL
LIN {X 0,Y 283.885,Z 507.474,A -85,B 0,C 180,E1 -17349.343,E2 -17349.343} C_VEL
LIN {X 0,Y 281.864,Z 516.167,A -85,B 0,C 180,E1 -17351.087,E2 -17351.087} C_VEL
LIN {X 0,Y 280.032,Z 524.736,A -85,B 0,C 180,E1 -17353.226,E2 -17353.226} C_VEL
LIN {X 0,Y 278.372,Z 531.664,A -85,B 0,C 180,E1 -17355.377,E2 -17355.377} C_VEL
LIN {X 0,Y 277.009,Z 537.258,A -85,B 0,C 180,E1 -17357.547,E2 -17357.547} C_VEL
LIN {X 0,Y 276.192,Z 541.685,A -85,B 0,C 180,E1 -17359.74,E2 -17359.74} C_VEL
LIN {X 0,Y 275.772,Z 544.048,A -85,B 0,C 180,E1 -17361.205,E2 -17361.205} C_VEL
LIN {X 0,Y 275.492,Z 545.986,A -85,B 0,C 180,E1 -17362.672,E2 -17362.672} C_VEL
LIN {X 0,Y 275.25,Z 548.535,A -85,B 0,C 180,E1 -17365.607,E2 -17365.607} C_VEL
LIN {X 0,Y 275.286,Z 549.221,A -85,B 0,C 180,E1 -17367.074,E2 -17367.074} C_VEL
LIN {X 0,Y 275.303,Z 549.513,A -85,B 0,C 180,E1 -17368.538,E2 -17368.538} C_VEL
LIN {X 0,Y 275.334,Z 549.364,A -85,B 0,C 180,E1 -17370.001,E2 -17370.001} C_VEL
LIN {X 0,Y 275.311,Z 548.804,A -85,B 0,C 180,E1 -17371.463,E2 -17371.463} C_VEL
LIN {X 0,Y 275.321,Z 547.846,A -85,B 0,C 180,E1 -17372.927,E2 -17372.927} C_VEL
LIN {X 0,Y 275.326,Z 545.227,A -85,B 0,C 180,E1 -17375.423,E2 -17375.423} C_VEL
LIN {X 0,Y 275.601,Z 540.997,A -85,B 0,C 180,E1 -17378.063,E2 -17378.063} C_VEL
LIN {X 0,Y 276.111,Z 536.236,A -85,B 0,C 180,E1 -17380.264,E2 -17380.264} C_VEL
LIN {X 0,Y 276.979,Z 529.064,A -85,B 0,C 180,E1 -17382.828,E2 -17382.828} C_VEL
LIN {X 0,Y 278.183,Z 521.243,A -85,B 0,C 180,E1 -17385.009,E2 -17385.009} C_VEL
LIN {X 0,Y 279.315,Z 514.077,A -85,B 0,C 180,E1 -17386.647,E2 -17386.647} C_VEL
LIN {X 0,Y 280.826,Z 503.52,A -85,B 0,C 180,E1 -17388.608,E2 -17388.608} C_VEL
LIN {X 0,Y 282.452,Z 492.774,A -85,B 0,C 180,E1 -17390.197,E2 -17390.197} C_VEL
LIN {X 0,Y 282.724,Z 488.514,A -85,B 0,C 180,E1 -17390.747,E2 -17390.747} C_VEL
LIN {X 0,Y 281.907,Z 477.62,A -85,B 0,C 180,E1 -17392.044,E2 -17392.044} C_VEL
LIN {X 0,Y 280.396,Z 464.931,A -85,B 0,C 180,E1 -17393.273,E2 -17393.273} C_VEL
LIN {X 0,Y 278.293,Z 451.753,A -85,B 0,C 180,E1 -17394.284,E2 -17394.284} C_VEL
LIN {X 0,Y 276.744,Z 443.37,A -85,B 0,C 180,E1 -17394.812,E2 -17394.812} C_VEL
LIN {X 0,Y 277.635,Z 436.785,A -85,B 0,C 180,E1 -17399.579,E2 -17399.579} C_VEL
LIN {X 0,Y 278.527,Z 431.209,A -85,B 0,C 180,E1 -17403.719,E2 -17403.719} C_VEL
LIN {X 0,Y 278.943,Z 427.873,A -85,B 0,C 180,E1 -17406.269,E2 -17406.269} C_VEL
LIN {X 0,Y 278.782,Z 424.388,A -85,B 0,C 180,E1 -17409.068,E2 -17409.068} C_VEL
LIN {X 0,Y 277.979,Z 419.947,A -85,B 0,C 180,E1 -17412.845,E2 -17412.845} C_VEL
LIN {X 0,Y 277.249,Z 415.951,A -85,B 0,C 180,E1 -17416.56,E2 -17416.56} C_VEL
LIN {X 0,Y 277.235,Z 415.953,A -85,B 0,C 180,E1 -17420.672,E2 -17420.672} C_VEL
LIN {X 0,Y 277.285,Z 415.939,A -85,B 0,C 180,E1 -17424.341,E2 -17424.341} C_VEL
LIN {X 0,Y 277.246,Z 415.949,A -85,B 0,C 180,E1 -17427.836,E2 -17427.836} C_VEL
LIN {X 0,Y 277.29,Z 415.943,A -85,B 0,C 180,E1 -17431.212,E2 -17431.212} C_VEL
LIN {X 0,Y 277.313,Z 415.937,A -85,B 0,C 180,E1 -17434.479,E2 -17434.479} C_VEL
LIN {X 0,Y 277.287,Z 415.944,A -85,B 0,C 180,E1 -17437.655,E2 -17437.655} C_VEL
LIN {X 0,Y 277.347,Z 415.937,A -85,B 0,C 180,E1 -17440.766,E2 -17440.766} C_VEL
LIN {X 0,Y 277.436,Z 415.926,A -85,B 0,C 180,E1 -17445.326,E2 -17445.326} C_VEL
LIN {X 0,Y 277.508,Z 415.914,A -85,B 0,C 180,E1 -17449.789,E2 -17449.789} C_VEL
LIN {X 0,Y 277.654,Z 415.899,A -85,B 0,C 180,E1 -17452.729,E2 -17452.729} C_VEL
LIN {X 0,Y 277.821,Z 415.876,A -85,B 0,C 180,E1 -17458.55,E2 -17458.55} C_VEL
LIN {X 0,Y 277.822,Z 415.876,A -85,B 0,C 180,E1 -17461.449,E2 -17461.449} C_VEL
LIN {X 0,Y 277.654,Z 415.898,A -85,B 0,C 180,E1 -17467.271,E2 -17467.271} C_VEL
LIN {X 0,Y 277.508,Z 415.915,A -85,B 0,C 180,E1 -17470.211,E2 -17470.211} C_VEL
LIN {X 0,Y 277.436,Z 415.924,A -85,B 0,C 180,E1 -17474.674,E2 -17474.674} C_VEL
LIN {X 0,Y 277.346,Z 415.93,A -85,B 0,C 180,E1 -17479.234,E2 -17479.234} C_VEL
LIN {X 0,Y 277.321,Z 415.937,A -85,B 0,C 180,E1 -17484.17,E2 -17484.17} C_VEL
LIN {X 0,Y 277.329,Z 415.937,A -85,B 0,C 180,E1 -17487.506,E2 -17487.506} C_VEL
LIN {X 0,Y 277.273,Z 415.946,A -85,B 0,C 180,E1 -17490.481,E2 -17490.481} C_VEL
LIN {X 0,Y 277.248,Z 415.942,A -85,B 0,C 180,E1 -17493.896,E2 -17493.896} C_VEL
LIN {X 0,Y 277.269,Z 415.939,A -85,B 0,C 180,E1 -17497.469,E2 -17497.469} C_VEL
LIN {X 0,Y 277.21,Z 415.952,A -85,B 0,C 180,E1 -17501.236,E2 -17501.236} C_VEL
LIN {X 0,Y 277.202,Z 415.953,A -85,B 0,C 180,E1 -17505.226,E2 -17505.226} C_VEL
LIN {X 0,Y 277.224,Z 415.946,A -85,B 0,C 180,E1 -17509.512,E2 -17509.512} C_VEL
LIN {X 0,Y 277.283,Z 415.942,A -85,B 0,C 180,E1 -17512.533,E2 -17512.533} C_VEL
LIN {X 0,Y 277.256,Z 415.947,A -85,B 0,C 180,E1 -17516.105,E2 -17516.105} C_VEL
LIN {X 0,Y 277.263,Z 415.945,A -85,B 0,C 180,E1 -17519.538,E2 -17519.538} C_VEL
LIN {X 0,Y 277.357,Z 415.932,A -85,B 0,C 180,E1 -17522.864,E2 -17522.864} C_VEL
LIN {X 0,Y 277.33,Z 415.938,A -85,B 0,C 180,E1 -17526.079,E2 -17526.079} C_VEL
LIN {X 0,Y 277.347,Z 415.935,A -85,B 0,C 180,E1 -17530.766,E2 -17530.766} C_VEL
LIN {X 0,Y 277.437,Z 415.924,A -85,B 0,C 180,E1 -17535.326,E2 -17535.326} C_VEL
LIN {X 0,Y 277.509,Z 415.915,A -85,B 0,C 180,E1 -17539.788,E2 -17539.788} C_VEL
LIN {X 0,Y 277.656,Z 415.898,A -85,B 0,C 180,E1 -17542.729,E2 -17542.729} C_VEL
LIN {X 0,Y 277.822,Z 415.88,A -85,B 0,C 180,E1 -17548.55,E2 -17548.55} C_VEL
LIN {X 0,Y 277.822,Z 415.876,A -85,B 0,C 180,E1 -17551.449,E2 -17551.449} C_VEL
LIN {X 0,Y 277.488,Z 415.92,A -85,B 0,C 180,E1 -17555.814,E2 -17555.814} C_VEL
LIN {X 0,Y 277.175,Z 415.959,A -85,B 0,C 180,E1 -17558.75,E2 -17558.75} C_VEL
LIN {X 0,Y 277.02,Z 416.139,A -85,B 0,C 180,E1 -17559.491,E2 -17559.491} C_VEL
LIN {X 0,Y 276.68,Z 419.458,A -85,B 0,C 180,E1 -17563.215,E2 -17563.215} C_VEL
LIN {X 0,Y 276.367,Z 422.191,A -85,B 0,C 180,E1 -17566.243,E2 -17566.243} C_VEL
LIN {X 0,Y 276.259,Z 424.141,A -85,B 0,C 180,E1 -17568.301,E2 -17568.301} C_VEL
LIN {X 0,Y 279.671,Z 437.593,A -85,B 0,C 180,E1 -17569.278,E2 -17569.278} C_VEL
LIN {X 0,Y 282.295,Z 449.696,A -85,B 0,C 180,E1 -17570.397,E2 -17570.397} C_VEL
LIN {X 0,Y 284.348,Z 461.804,A -85,B 0,C 180,E1 -17571.761,E2 -17571.761} C_VEL
LIN {X 0,Y 282.968,Z 473.709,A -85,B 0,C 180,E1 -17573.225,E2 -17573.225} C_VEL
LIN {X 0,Y 281.434,Z 484.695,A -85,B 0,C 180,E1 -17574.922,E2 -17574.922} C_VEL
LIN {X 0,Y 279.879,Z 494.681,A -85,B 0,C 180,E1 -17576.871,E2 -17576.871} C_VEL
LIN {X 0,Y 278.501,Z 503.671,A -85,B 0,C 180,E1 -17579.062,E2 -17579.062} C_VEL
LIN {X 0,Y 277.337,Z 511.067,A -85,B 0,C 180,E1 -17581.348,E2 -17581.348} C_VEL
LIN {X 0,Y 276.506,Z 516.556,A -85,B 0,C 180,E1 -17583.48,E2 -17583.48} C_VEL
LIN {X 0,Y 275.874,Z 521.329,A -85,B 0,C 180,E1 -17585.868,E2 -17585.868} C_VEL
LIN {X 0,Y 275.328,Z 525.378,A -85,B 0,C 180,E1 -17588.709,E2 -17588.709} C_VEL
LIN {X 0,Y 275.167,Z 526.637,A -85,B 0,C 180,E1 -17589.984,E2 -17589.984} C_VEL
LIN {X 0,Y 275.044,Z 528.098,A -85,B 0,C 180,E1 -17592.182,E2 -17592.182} C_VEL
LIN {X 0,Y 275.033,Z 528.641,A -85,B 0,C 180,E1 -17594.316,E2 -17594.316} C_VEL
LIN {X 0,Y 275.231,Z 528.336,A -85,B 0,C 180,E1 -17596.414,E2 -17596.414} C_VEL
LIN {X 0,Y 275.585,Z 527.261,A -85,B 0,C 180,E1 -17598.467,E2 -17598.467} C_VEL
LIN {X 0,Y 276.138,Z 525.439,A -85,B 0,C 180,E1 -17600.485,E2 -17600.485} C_VEL
LIN {X 0,Y 277.227,Z 521.419,A -85,B 0,C 180,E1 -17603.351,E2 -17603.351} C_VEL
LIN {X 0,Y 278.54,Z 516.438,A -85,B 0,C 180,E1 -17605.848,E2 -17605.848} C_VEL
LIN {X 0,Y 280.152,Z 510.178,A -85,B 0,C 180,E1 -17608.21,E2 -17608.21} C_VEL
LIN {X 0,Y 282.034,Z 502.756,A -85,B 0,C 180,E1 -17610.416,E2 -17610.416} C_VEL
LIN {X 0,Y 284.148,Z 494.346,A -85,B 0,C 180,E1 -17612.409,E2 -17612.409} C_VEL
LIN {X 0,Y 286.088,Z 485.793,A -85,B 0,C 180,E1 -17614.052,E2 -17614.052} C_VEL
LIN {X 0,Y 288.209,Z 475.15,A -85,B 0,C 180,E1 -17615.701,E2 -17615.701} C_VEL
LIN {X 0,Y 289.361,Z 468.527,A -85,B 0,C 180,E1 -17616.565,E2 -17616.565} C_VEL
LIN {X 0,Y 287.914,Z 458.394,A -85,B 0,C 180,E1 -17618.031,E2 -17618.031} C_VEL
LIN {X 0,Y 285.256,Z 447.533,A -85,B 0,C 180,E1 -17619.505,E2 -17619.505} C_VEL
LIN {X 0,Y 281.254,Z 436.129,A -85,B 0,C 180,E1 -17620.979,E2 -17620.979} C_VEL
LIN {X 0,Y 278.312,Z 429.392,A -85,B 0,C 180,E1 -17621.838,E2 -17621.838} C_VEL
LIN {X 0,Y 277.304,Z 426.312,A -85,B 0,C 180,E1 -17622.199,E2 -17622.199} C_VEL
LIN {X 0,Y 277.679,Z 424.032,A -85,B 0,C 180,E1 -17625.339,E2 -17625.339} C_VEL
LIN {X 0,Y 277.99,Z 422.005,A -85,B 0,C 180,E1 -17628.331,E2 -17628.331} C_VEL
LIN {X 0,Y 278.197,Z 420.136,A -85,B 0,C 180,E1 -17631.282,E2 -17631.282} C_VEL
LIN {X 0,Y 277.983,Z 418.513,A -85,B 0,C 180,E1 -17634.196,E2 -17634.196} C_VEL
LIN {X 0,Y 277.879,Z 416.336,A -85,B 0,C 180,E1 -17638.551,E2 -17638.551} C_VEL
LIN {X 0,Y 277.891,Z 415.871,A -85,B 0,C 180,E1 -17640,E2 -17640} C_VEL
LIN {X 0,Y 277.697,Z 415.894,A -85,B 0,C 180,E1 -17642.901,E2 -17642.901} C_VEL
LIN {X 0,Y 277.535,Z 415.914,A -85,B 0,C 180,E1 -17645.543,E2 -17645.543} C_VEL
LIN {X 0,Y 276.946,Z 415.99,A -85,B 0,C 180,E1 -17646.755,E2 -17646.755} C_VEL
LIN {X 0,Y 274.039,Z 416.351,A -85,B 0,C 180,E1 -17648.727,E2 -17648.727} C_VEL
LIN {X 0,Y 271.528,Z 416.663,A -85,B 0,C 180,E1 -17650.331,E2 -17650.331} C_VEL
LIN {X 0,Y 270.467,Z 416.796,A -85,B 0,C 180,E1 -17651.576,E2 -17651.576} C_VEL
LIN {X 0,Y 270.395,Z 416.804,A -85,B 0,C 180,E1 -17651.998,E2 -17651.998} C_VEL
LIN {X 0,Y 270.377,Z 416.806,A -85,B 0,C 180,E1 -17655.901,E2 -17655.901} C_VEL
LIN {X 0,Y 270.289,Z 416.818,A -85,B 0,C 180,E1 -17660.602,E2 -17660.602} C_VEL
LIN {X 0,Y 270.271,Z 416.815,A -85,B 0,C 180,E1 -17664.586,E2 -17664.586} C_VEL
LIN {X 0,Y 270.269,Z 416.82,A -85,B 0,C 180,E1 -17667.909,E2 -17667.909} C_VEL
LIN {X 0,Y 270.222,Z 416.949,A -85,B 0,C 180,E1 -17671.344,E2 -17671.344} C_VEL
LIN {X 0,Y 270.533,Z 418.631,A -85,B 0,C 180,E1 -17674.857,E2 -17674.857} C_VEL
LIN {X 0,Y 270.956,Z 421.025,A -85,B 0,C 180,E1 -17678.912,E2 -17678.912} C_VEL
LIN {X 0,Y 271.353,Z 423.415,A -85,B 0,C 180,E1 -17682.33,E2 -17682.33} C_VEL
LIN {X 0,Y 271.886,Z 426.67,A -85,B 0,C 180,E1 -17686.367,E2 -17686.367} C_VEL
LIN {X 0,Y 272.348,Z 429.8,A -85,B 0,C 180,E1 -17689.826,E2 -17689.826} C_VEL
LIN {X 0,Y 272.567,Z 433.056,A -85,B 0,C 180,E1 -17693.066,E2 -17693.066} C_VEL
LIN {X 0,Y 272.144,Z 436.034,A -85,B 0,C 180,E1 -17695.73,E2 -17695.73} C_VEL
LIN {X 0,Y 271.081,Z 440.937,A -85,B 0,C 180,E1 -17699.835,E2 -17699.835} C_VEL
LIN {X 0,Y 271.963,Z 444.164,A -85,B 0,C 180,E1 -17700.147,E2 -17700.147} C_VEL
LIN {X 0,Y 275.293,Z 454.164,A -85,B 0,C 180,E1 -17701.307,E2 -17701.307} C_VEL
LIN {X 0,Y 278.101,Z 465.741,A -85,B 0,C 180,E1 -17702.678,E2 -17702.678} C_VEL
LIN {X 0,Y 279.624,Z 476.12,A -85,B 0,C 180,E1 -17703.984,E2 -17703.984} C_VEL
LIN {X 0,Y 280.292,Z 487.061,A -85,B 0,C 180,E1 -17705.499,E2 -17705.499} C_VEL
LIN {X 0,Y 279.999,Z 496.366,A -85,B 0,C 180,E1 -17706.91,E2 -17706.91} C_VEL
LIN {X 0,Y 277.749,Z 506.032,A -85,B 0,C 180,E1 -17708.476,E2 -17708.476} C_VEL
LIN {X 0,Y 275.559,Z 514.911,A -85,B 0,C 180,E1 -17710.25,E2 -17710.25} C_VEL
LIN {X 0,Y 273.464,Z 523.66,A -85,B 0,C 180,E1 -17712.425,E2 -17712.425} C_VEL
LIN {X 0,Y 271.77,Z 530.728,A -85,B 0,C 180,E1 -17714.63,E2 -17714.63} C_VEL
LIN {X 0,Y 270.046,Z 537.259,A -85,B 0,C 180,E1 -17717.22,E2 -17717.22} C_VEL
LIN {X 0,Y 269.192,Z 541.623,A -85,B 0,C 180,E1 -17719.47,E2 -17719.47} C_VEL
LIN {X 0,Y 268.728,Z 543.956,A -85,B 0,C 180,E1 -17720.973,E2 -17720.973} C_VEL
LIN {X 0,Y 268.416,Z 545.845,A -85,B 0,C 180,E1 -17722.478,E2 -17722.478} C_VEL
LIN {X 0,Y 268.165,Z 548.328,A -85,B 0,C 180,E1 -17725.491,E2 -17725.491} C_VEL
LIN {X 0,Y 268.195,Z 548.986,A -85,B 0,C 180,E1 -17726.996,E2 -17726.996} C_VEL
LIN {X 0,Y 268.226,Z 549.235,A -85,B 0,C 180,E1 -17728.499,E2 -17728.499} C_VEL
LIN {X 0,Y 268.256,Z 549.048,A -85,B 0,C 180,E1 -17730.001,E2 -17730.001} C_VEL
LIN {X 0,Y 268.236,Z 548.464,A -85,B 0,C 180,E1 -17731.502,E2 -17731.502} C_VEL
LIN {X 0,Y 268.229,Z 547.48,A -85,B 0,C 180,E1 -17733.004,E2 -17733.004} C_VEL
LIN {X 0,Y 268.225,Z 545.09,A -85,B 0,C 180,E1 -17735.33,E2 -17735.33} C_VEL
LIN {X 0,Y 268.438,Z 541.847,A -85,B 0,C 180,E1 -17737.522,E2 -17737.522} C_VEL
LIN {X 0,Y 268.881,Z 537.421,A -85,B 0,C 180,E1 -17739.782,E2 -17739.782} C_VEL
LIN {X 0,Y 269.511,Z 531.764,A -85,B 0,C 180,E1 -17742.042,E2 -17742.042} C_VEL
LIN {X 0,Y 270.666,Z 524.684,A -85,B 0,C 180,E1 -17744.281,E2 -17744.281} C_VEL
LIN {X 0,Y 272.092,Z 515.829,A -85,B 0,C 180,E1 -17746.507,E2 -17746.507} C_VEL
LIN {X 0,Y 273.419,Z 506.753,A -85,B 0,C 180,E1 -17748.354,E2 -17748.354} C_VEL
LIN {X 0,Y 274.915,Z 496.787,A -85,B 0,C 180,E1 -17749.994,E2 -17749.994} C_VEL
LIN {X 0,Y 275.821,Z 490.181,A -85,B 0,C 180,E1 -17750.9,E2 -17750.9} C_VEL
LIN {X 0,Y 275.109,Z 479.359,A -85,B 0,C 180,E1 -17752.266,E2 -17752.266} C_VEL
LIN {X 0,Y 273.674,Z 466.593,A -85,B 0,C 180,E1 -17753.587,E2 -17753.587} C_VEL
LIN {X 0,Y 271.539,Z 452.982,A -85,B 0,C 180,E1 -17754.688,E2 -17754.688} C_VEL
LIN {X 0,Y 269.719,Z 443.166,A -85,B 0,C 180,E1 -17755.316,E2 -17755.316} C_VEL
LIN {X 0,Y 270.563,Z 437.452,A -85,B 0,C 180,E1 -17759.573,E2 -17759.573} C_VEL
LIN {X 0,Y 271.557,Z 431.526,A -85,B 0,C 180,E1 -17764.088,E2 -17764.088} C_VEL
LIN {X 0,Y 271.894,Z 428.175,A -85,B 0,C 180,E1 -17766.745,E2 -17766.745} C_VEL
LIN {X 0,Y 271.743,Z 425.298,A -85,B 0,C 180,E1 -17769.115,E2 -17769.115} C_VEL
LIN {X 0,Y 271.064,Z 421.55,A -85,B 0,C 180,E1 -17772.386,E2 -17772.386} C_VEL
LIN {X 0,Y 270.195,Z 416.83,A -85,B 0,C 180,E1 -17776.745,E2 -17776.745} C_VEL
LIN {X 0,Y 270.209,Z 416.828,A -85,B 0,C 180,E1 -17781.374,E2 -17781.374} C_VEL
LIN {X 0,Y 270.203,Z 416.826,A -85,B 0,C 180,E1 -17785.094,E2 -17785.094} C_VEL
LIN {X 0,Y 270.202,Z 416.83,A -85,B 0,C 180,E1 -17789.131,E2 -17789.131} C_VEL
LIN {X 0,Y 270.266,Z 416.813,A -85,B 0,C 180,E1 -17792.146,E2 -17792.146} C_VEL
LIN {X 0,Y 270.279,Z 416.816,A -85,B 0,C 180,E1 -17795.519,E2 -17795.519} C_VEL
LIN {X 0,Y 270.303,Z 416.812,A -85,B 0,C 180,E1 -17800.244,E2 -17800.244} C_VEL
LIN {X 0,Y 270.405,Z 416.803,A -85,B 0,C 180,E1 -17804.935,E2 -17804.935} C_VEL
LIN {X 0,Y 270.443,Z 416.795,A -85,B 0,C 180,E1 -17809.519,E2 -17809.519} C_VEL
LIN {X 0,Y 270.613,Z 416.775,A -85,B 0,C 180,E1 -17812.539,E2 -17812.539} C_VEL
LIN {X 0,Y 270.787,Z 416.752,A -85,B 0,C 180,E1 -17818.513,E2 -17818.513} C_VEL
LIN {X 0,Y 270.788,Z 416.752,A -85,B 0,C 180,E1 -17821.487,E2 -17821.487} C_VEL
LIN {X 0,Y 270.612,Z 416.774,A -85,B 0,C 180,E1 -17827.461,E2 -17827.461} C_VEL
LIN {X 0,Y 270.443,Z 416.796,A -85,B 0,C 180,E1 -17830.481,E2 -17830.481} C_VEL
LIN {X 0,Y 270.404,Z 416.796,A -85,B 0,C 180,E1 -17835.064,E2 -17835.064} C_VEL
LIN {X 0,Y 270.303,Z 416.805,A -85,B 0,C 180,E1 -17839.755,E2 -17839.755} C_VEL
LIN {X 0,Y 270.276,Z 416.817,A -85,B 0,C 180,E1 -17844.585,E2 -17844.585} C_VEL
LIN {X 0,Y 270.274,Z 416.816,A -85,B 0,C 180,E1 -17847.908,E2 -17847.908} C_VEL
LIN {X 0,Y 270.186,Z 416.825,A -85,B 0,C 180,E1 -17851.348,E2 -17851.348} C_VEL
LIN {X 0,Y 270.203,Z 416.817,A -85,B 0,C 180,E1 -17854.905,E2 -17854.905} C_VEL
LIN {X 0,Y 270.199,Z 416.825,A -85,B 0,C 180,E1 -17858.71,E2 -17858.71} C_VEL
LIN {X 0,Y 270.173,Z 416.832,A -85,B 0,C 180,E1 -17862.558,E2 -17862.558} C_VEL
LIN {X 0,Y 270.166,Z 416.831,A -85,B 0,C 180,E1 -17866.751,E2 -17866.751} C_VEL
LIN {X 0,Y 270.224,Z 416.816,A -85,B 0,C 180,E1 -17871.283,E2 -17871.283} C_VEL
LIN {X 0,Y 270.216,Z 416.823,A -85,B 0,C 180,E1 -17875.096,E2 -17875.096} C_VEL
LIN {X 0,Y 270.202,Z 416.825,A -85,B 0,C 180,E1 -17879.13,E2 -17879.13} C_VEL
LIN {X 0,Y 270.265,Z 416.816,A -85,B 0,C 180,E1 -17882.146,E2 -17882.146} C_VEL
LIN {X 0,Y 270.279,Z 416.814,A -85,B 0,C 180,E1 -17885.519,E2 -17885.519} C_VEL
LIN {X 0,Y 270.304,Z 416.815,A -85,B 0,C 180,E1 -17890.244,E2 -17890.244} C_VEL
LIN {X 0,Y 270.405,Z 416.802,A -85,B 0,C 180,E1 -17894.935,E2 -17894.935} C_VEL
LIN {X 0,Y 270.444,Z 416.794,A -85,B 0,C 180,E1 -17899.519,E2 -17899.519} C_VEL
LIN {X 0,Y 270.614,Z 416.776,A -85,B 0,C 180,E1 -17902.538,E2 -17902.538} C_VEL
LIN {X 0,Y 270.788,Z 416.756,A -85,B 0,C 180,E1 -17908.512,E2 -17908.512} C_VEL
LIN {X 0,Y 270.788,Z 416.753,A -85,B 0,C 180,E1 -17911.487,E2 -17911.487} C_VEL
LIN {X 0,Y 270.447,Z 416.799,A -85,B 0,C 180,E1 -17915.966,E2 -17915.966} C_VEL
LIN {X 0,Y 270.011,Z 416.851,A -85,B 0,C 180,E1 -17919.173,E2 -17919.173} C_VEL
LIN {X 0,Y 269.598,Z 420.617,A -85,B 0,C 180,E1 -17923.568,E2 -17923.568} C_VEL
LIN {X 0,Y 269.2,Z 424.092,A -85,B 0,C 180,E1 -17927.471,E2 -17927.471} C_VEL
LIN {X 0,Y 269.2,Z 424.413,A -85,B 0,C 180,E1 -17927.765,E2 -17927.765} C_VEL
LIN {X 0,Y 272.576,Z 437.534,A -85,B 0,C 180,E1 -17928.752,E2 -17928.752} C_VEL
LIN {X 0,Y 275.349,Z 450.224,A -85,B 0,C 180,E1 -17929.96,E2 -17929.96} C_VEL
LIN {X 0,Y 277.392,Z 462.28,A -85,B 0,C 180,E1 -17931.358,E2 -17931.358} C_VEL
LIN {X 0,Y 277.25,Z 465.621,A -85,B 0,C 180,E1 -17931.76,E2 -17931.76} C_VEL
LIN {X 0,Y 275.913,Z 475.8,A -85,B 0,C 180,E1 -17933.102,E2 -17933.102} C_VEL
LIN {X 0,Y 274.374,Z 486.137,A -85,B 0,C 180,E1 -17934.798,E2 -17934.798} C_VEL
LIN {X 0,Y 272.788,Z 495.928,A -85,B 0,C 180,E1 -17936.798,E2 -17936.798} C_VEL
LIN {X 0,Y 271.459,Z 504.26,A -85,B 0,C 180,E1 -17938.914,E2 -17938.914} C_VEL
LIN {X 0,Y 270.245,Z 511.804,A -85,B 0,C 180,E1 -17941.339,E2 -17941.339} C_VEL
LIN {X 0,Y 269.418,Z 516.945,A -85,B 0,C 180,E1 -17943.411,E2 -17943.411} C_VEL
LIN {X 0,Y 268.779,Z 521.666,A -85,B 0,C 180,E1 -17945.847,E2 -17945.847} C_VEL
LIN {X 0,Y 268.303,Z 525.033,A -85,B 0,C 180,E1 -17948.203,E2 -17948.203} C_VEL
LIN {X 0,Y 268.006,Z 527.634,A -85,B 0,C 180,E1 -17950.963,E2 -17950.963} C_VEL
LIN {X 0,Y 267.917,Z 528.628,A -85,B 0,C 180,E1 -17953.001,E2 -17953.001} C_VEL
LIN {X 0,Y 267.974,Z 528.906,A -85,B 0,C 180,E1 -17955.08,E2 -17955.08} C_VEL
LIN {X 0,Y 268.248,Z 528.429,A -85,B 0,C 180,E1 -17957.187,E2 -17957.187} C_VEL
LIN {X 0,Y 268.708,Z 527.128,A -85,B 0,C 180,E1 -17959.33,E2 -17959.33} C_VEL
LIN {X 0,Y 269.721,Z 523.793,A -85,B 0,C 180,E1 -17962.375,E2 -17962.375} C_VEL
LIN {X 0,Y 271.094,Z 519.034,A -85,B 0,C 180,E1 -17965.226,E2 -17965.226} C_VEL
LIN {X 0,Y 272.671,Z 513.269,A -85,B 0,C 180,E1 -17967.73,E2 -17967.73} C_VEL
LIN {X 0,Y 274.339,Z 507.183,A -85,B 0,C 180,E1 -17969.807,E2 -17969.807} C_VEL
LIN {X 0,Y 276.364,Z 499.713,A -85,B 0,C 180,E1 -17971.856,E2 -17971.856} C_VEL
LIN {X 0,Y 278.612,Z 490.898,A -85,B 0,C 180,E1 -17973.804,E2 -17973.804} C_VEL
LIN {X 0,Y 280.913,Z 480.603,A -85,B 0,C 180,E1 -17975.619,E2 -17975.619} C_VEL
LIN {X 0,Y 282.97,Z 470.112,A -85,B 0,C 180,E1 -17977.099,E2 -17977.099} C_VEL
LIN {X 0,Y 281.536,Z 459.891,A -85,B 0,C 180,E1 -17978.678,E2 -17978.678} C_VEL
LIN {X 0,Y 278.811,Z 448.63,A -85,B 0,C 180,E1 -17980.297,E2 -17980.297} C_VEL
LIN {X 0,Y 274.639,Z 436.89,A -85,B 0,C 180,E1 -17981.924,E2 -17981.924} C_VEL
LIN {X 0,Y 271.418,Z 429.682,A -85,B 0,C 180,E1 -17982.919,E2 -17982.919} C_VEL
LIN {X 0,Y 270.416,Z 426.687,A -85,B 0,C 180,E1 -17983.267,E2 -17983.267} C_VEL
LIN {X 0,Y 270.797,Z 424.475,A -85,B 0,C 180,E1 -17986.492,E2 -17986.492} C_VEL
LIN {X 0,Y 271.137,Z 422.202,A -85,B 0,C 180,E1 -17990.05,E2 -17990.05} C_VEL
LIN {X 0,Y 271.162,Z 420.745,A -85,B 0,C 180,E1 -17992.554,E2 -17992.554} C_VEL
LIN {X 0,Y 270.906,Z 418.507,A -85,B 0,C 180,E1 -17997.026,E2 -17997.026} C_VEL
LIN {X 0,Y 270.926,Z 417.173,A -85,B 0,C 180,E1 -18000,E2 -18000} C_VEL
LIN {X 0,Y 270.785,Z 416.756,A -85,B 0,C 180,E1 -18001.487,E2 -18001.487} C_VEL
LIN {X 0,Y 270.608,Z 416.779,A -85,B 0,C 180,E1 -18007.461,E2 -18007.461} C_VEL
LIN {X 0,Y 270.438,Z 416.799,A -85,B 0,C 180,E1 -18010.481,E2 -18010.481} C_VEL
LIN {X 0,Y 270.395,Z 416.804,A -85,B 0,C 180,E1 -18011.998,E2 -18011.998} C_VEL
LIN {X 0,Y 269.741,Z 416.891,A -85,B 0,C 180,E1 -18013.243,E2 -18013.243} C_VEL
LIN {X 0,Y 266.819,Z 417.251,A -85,B 0,C 180,E1 -18015.267,E2 -18015.267} C_VEL
LIN {X 0,Y 264.342,Z 417.558,A -85,B 0,C 180,E1 -18016.914,E2 -18016.914} C_VEL
LIN {X 0,Y 263.309,Z 417.687,A -85,B 0,C 180,E1 -18018.193,E2 -18018.193} C_VEL
LIN {X 0,Y 263.244,Z 417.694,A -85,B 0,C 180,E1 -18018.626,E2 -18018.626} C_VEL
LIN {X 0,Y 263.155,Z 417.706,A -85,B 0,C 180,E1 -18021.956,E2 -18021.956} C_VEL
LIN {X 0,Y 263.206,Z 417.7,A -85,B 0,C 180,E1 -18025.292,E2 -18025.292} C_VEL
LIN {X 0,Y 263.177,Z 417.704,A -85,B 0,C 180,E1 -18028.73,E2 -18028.73} C_VEL
LIN {X 0,Y 263.363,Z 419.03,A -85,B 0,C 180,E1 -18032.257,E2 -18032.257} C_VEL
LIN {X 0,Y 263.715,Z 420.824,A -85,B 0,C 180,E1 -18035.895,E2 -18035.895} C_VEL
LIN {X 0,Y 264.134,Z 423.096,A -85,B 0,C 180,E1 -18039.687,E2 -18039.687} C_VEL
LIN {X 0,Y 264.663,Z 426.344,A -85,B 0,C 180,E1 -18044.196,E2 -18044.196} C_VEL
LIN {X 0,Y 265.138,Z 429.417,A -85,B 0,C 180,E1 -18047.919,E2 -18047.919} C_VEL
LIN {X 0,Y 265.453,Z 431.814,A -85,B 0,C 180,E1 -18050.551,E2 -18050.551} C_VEL
LIN {X 0,Y 265.557,Z 433.792,A -85,B 0,C 180,E1 -18052.557,E2 -18052.557} C_VEL
LIN {X 0,Y 265.229,Z 436.636,A -85,B 0,C 180,E1 -18055.229,E2 -18055.229} C_VEL
LIN {X 0,Y 264.349,Z 440.746,A -85,B 0,C 180,E1 -18058.702,E2 -18058.702} C_VEL
LIN {X 0,Y 265.305,Z 444.001,A -85,B 0,C 180,E1 -18059.046,E2 -18059.046} C_VEL
LIN {X 0,Y 268.388,Z 453.094,A -85,B 0,C 180,E1 -18060.164,E2 -18060.164} C_VEL
LIN {X 0,Y 271.204,Z 463.831,A -85,B 0,C 180,E1 -18061.531,E2 -18061.531} C_VEL
LIN {X 0,Y 273.189,Z 476.19,A -85,B 0,C 180,E1 -18063.165,E2 -18063.165} C_VEL
LIN {X 0,Y 273.837,Z 486.31,A -85,B 0,C 180,E1 -18064.614,E2 -18064.614} C_VEL
LIN {X 0,Y 273.634,Z 495.936,A -85,B 0,C 180,E1 -18066.14,E2 -18066.14} C_VEL
LIN {X 0,Y 271.695,Z 504.608,A -85,B 0,C 180,E1 -18067.572,E2 -18067.572} C_VEL
LIN {X 0,Y 269.349,Z 513.654,A -85,B 0,C 180,E1 -18069.376,E2 -18069.376} C_VEL
LIN {X 0,Y 267.051,Z 522.563,A -85,B 0,C 180,E1 -18071.591,E2 -18071.591} C_VEL
LIN {X 0,Y 265.235,Z 529.801,A -85,B 0,C 180,E1 -18073.847,E2 -18073.847} C_VEL
LIN {X 0,Y 263.534,Z 535.648,A -85,B 0,C 180,E1 -18076.113,E2 -18076.113} C_VEL
LIN {X 0,Y 262.441,Z 540.293,A -85,B 0,C 180,E1 -18078.414,E2 -18078.414} C_VEL
LIN {X 0,Y 261.704,Z 543.867,A -85,B 0,C 180,E1 -18080.728,E2 -18080.728} C_VEL
LIN {X 0,Y 261.351,Z 545.694,A -85,B 0,C 180,E1 -18082.274,E2 -18082.274} C_VEL
LIN {X 0,Y 261.067,Z 548.122,A -85,B 0,C 180,E1 -18085.368,E2 -18085.368} C_VEL
LIN {X 0,Y 261.107,Z 548.751,A -85,B 0,C 180,E1 -18086.915,E2 -18086.915} C_VEL
LIN {X 0,Y 261.152,Z 548.945,A -85,B 0,C 180,E1 -18088.458,E2 -18088.458} C_VEL
LIN {X 0,Y 261.179,Z 548.729,A -85,B 0,C 180,E1 -18090.001,E2 -18090.001} C_VEL
LIN {X 0,Y 261.161,Z 548.116,A -85,B 0,C 180,E1 -18091.543,E2 -18091.543} C_VEL
LIN {X 0,Y 261.139,Z 547.101,A -85,B 0,C 180,E1 -18093.086,E2 -18093.086} C_VEL
LIN {X 0,Y 261.125,Z 544.931,A -85,B 0,C 180,E1 -18095.231,E2 -18095.231} C_VEL
LIN {X 0,Y 261.364,Z 541.339,A -85,B 0,C 180,E1 -18097.727,E2 -18097.727} C_VEL
LIN {X 0,Y 261.835,Z 536.844,A -85,B 0,C 180,E1 -18100.048,E2 -18100.048} C_VEL
LIN {X 0,Y 262.717,Z 529.992,A -85,B 0,C 180,E1 -18102.75,E2 -18102.75} C_VEL
LIN {X 0,Y 263.944,Z 522.544,A -85,B 0,C 180,E1 -18105.047,E2 -18105.047} C_VEL
LIN {X 0,Y 265.376,Z 513.788,A -85,B 0,C 180,E1 -18107.215,E2 -18107.215} C_VEL
LIN {X 0,Y 266.958,Z 503.635,A -85,B 0,C 180,E1 -18109.213,E2 -18109.213} C_VEL
LIN {X 0,Y 268.668,Z 493.034,A -85,B 0,C 180,E1 -18110.88,E2 -18110.88} C_VEL
LIN {X 0,Y 268.772,Z 487.475,A -85,B 0,C 180,E1 -18111.659,E2 -18111.659} C_VEL
LIN {X 0,Y 267.701,Z 474.977,A -85,B 0,C 180,E1 -18113.191,E2 -18113.191} C_VEL
LIN {X 0,Y 266.093,Z 461.963,A -85,B 0,C 180,E1 -18114.48,E2 -18114.48} C_VEL
LIN {X 0,Y 263.829,Z 448.838,A -85,B 0,C 180,E1 -18115.496,E2 -18115.496} C_VEL
LIN {X 0,Y 262.724,Z 442.958,A -85,B 0,C 180,E1 -18115.862,E2 -18115.862} C_VEL
LIN {X 0,Y 263.656,Z 436.989,A -85,B 0,C 180,E1 -18120.429,E2 -18120.429} C_VEL
LIN {X 0,Y 264.613,Z 431.712,A -85,B 0,C 180,E1 -18124.579,E2 -18124.579} C_VEL
LIN {X 0,Y 264.814,Z 428.471,A -85,B 0,C 180,E1 -18127.233,E2 -18127.233} C_VEL
LIN {X 0,Y 264.614,Z 425.676,A -85,B 0,C 180,E1 -18129.626,E2 -18129.626} C_VEL
LIN {X 0,Y 263.708,Z 420.864,A -85,B 0,C 180,E1 -18133.981,E2 -18133.981} C_VEL
LIN {X 0,Y 263.154,Z 417.708,A -85,B 0,C 180,E1 -18137.095,E2 -18137.095} C_VEL
LIN {X 0,Y 263.16,Z 417.703,A -85,B 0,C 180,E1 -18142.103,E2 -18142.103} C_VEL
LIN {X 0,Y 263.153,Z 417.704,A -85,B 0,C 180,E1 -18145.885,E2 -18145.885} C_VEL
LIN {X 0,Y 263.152,Z 417.705,A -85,B 0,C 180,E1 -18149.507,E2 -18149.507} C_VEL
LIN {X 0,Y 263.194,Z 417.696,A -85,B 0,C 180,E1 -18153.003,E2 -18153.003} C_VEL
LIN {X 0,Y 263.186,Z 417.699,A -85,B 0,C 180,E1 -18156.387,E2 -18156.387} C_VEL
LIN {X 0,Y 263.265,Z 417.689,A -85,B 0,C 180,E1 -18159.693,E2 -18159.693} C_VEL
LIN {X 0,Y 263.353,Z 417.679,A -85,B 0,C 180,E1 -18164.522,E2 -18164.522} C_VEL
LIN {X 0,Y 263.376,Z 417.677,A -85,B 0,C 180,E1 -18169.234,E2 -18169.234} C_VEL
LIN {X 0,Y 263.574,Z 417.651,A -85,B 0,C 180,E1 -18172.338,E2 -18172.338} C_VEL
LIN {X 0,Y 263.752,Z 417.628,A -85,B 0,C 180,E1 -18178.473,E2 -18178.473} C_VEL
LIN {X 0,Y 263.752,Z 417.628,A -85,B 0,C 180,E1 -18181.527,E2 -18181.527} C_VEL
LIN {X 0,Y 263.574,Z 417.65,A -85,B 0,C 180,E1 -18187.661,E2 -18187.661} C_VEL
LIN {X 0,Y 263.376,Z 417.678,A -85,B 0,C 180,E1 -18190.765,E2 -18190.765} C_VEL
LIN {X 0,Y 263.352,Z 417.671,A -85,B 0,C 180,E1 -18195.478,E2 -18195.478} C_VEL
LIN {X 0,Y 263.265,Z 417.682,A -85,B 0,C 180,E1 -18200.306,E2 -18200.306} C_VEL
LIN {X 0,Y 263.211,Z 417.697,A -85,B 0,C 180,E1 -18205.291,E2 -18205.291} C_VEL
LIN {X 0,Y 263.182,Z 417.703,A -85,B 0,C 180,E1 -18208.729,E2 -18208.729} C_VEL
LIN {X 0,Y 263.134,Z 417.704,A -85,B 0,C 180,E1 -18212.288,E2 -18212.288} C_VEL
LIN {X 0,Y 263.184,Z 417.693,A -85,B 0,C 180,E1 -18216.763,E2 -18216.763} C_VEL
LIN {X 0,Y 263.125,Z 417.705,A -85,B 0,C 180,E1 -18221.593,E2 -18221.593} C_VEL
LIN {X 0,Y 263.106,Z 417.71,A -85,B 0,C 180,E1 -18226.155,E2 -18226.155} C_VEL
LIN {X 0,Y 263.116,Z 417.703,A -85,B 0,C 180,E1 -18230.129,E2 -18230.129} C_VEL
LIN {X 0,Y 263.189,Z 417.696,A -85,B 0,C 180,E1 -18234.022,E2 -18234.022} C_VEL
LIN {X 0,Y 263.135,Z 417.706,A -85,B 0,C 180,E1 -18237.712,E2 -18237.712} C_VEL
LIN {X 0,Y 263.2,Z 417.695,A -85,B 0,C 180,E1 -18241.784,E2 -18241.784} C_VEL
LIN {X 0,Y 263.227,Z 417.693,A -85,B 0,C 180,E1 -18245.2,E2 -18245.2} C_VEL
LIN {X 0,Y 263.266,Z 417.689,A -85,B 0,C 180,E1 -18249.693,E2 -18249.693} C_VEL
LIN {X 0,Y 263.353,Z 417.683,A -85,B 0,C 180,E1 -18254.522,E2 -18254.522} C_VEL
LIN {X 0,Y 263.376,Z 417.674,A -85,B 0,C 180,E1 -18259.234,E2 -18259.234} C_VEL
LIN {X 0,Y 263.576,Z 417.655,A -85,B 0,C 180,E1 -18262.338,E2 -18262.338} C_VEL
LIN {X 0,Y 263.752,Z 417.633,A -85,B 0,C 180,E1 -18268.473,E2 -18268.473} C_VEL
LIN {X 0,Y 263.752,Z 417.63,A -85,B 0,C 180,E1 -18271.526,E2 -18271.526} C_VEL
LIN {X 0,Y 263.403,Z 417.678,A -85,B 0,C 180,E1 -18276.126,E2 -18276.126} C_VEL
LIN {X 0,Y 262.956,Z 417.73,A -85,B 0,C 180,E1 -18279.227,E2 -18279.227} C_VEL
LIN {X 0,Y 262.493,Z 421.749,A -85,B 0,C 180,E1 -18283.943,E2 -18283.943} C_VEL
LIN {X 0,Y 262.17,Z 424.67,A -85,B 0,C 180,E1 -18287.2,E2 -18287.2} C_VEL
LIN {X 0,Y 265.663,Z 438.138,A -85,B 0,C 180,E1 -18288.259,E2 -18288.259} C_VEL
LIN {X 0,Y 268.406,Z 450.704,A -85,B 0,C 180,E1 -18289.502,E2 -18289.502} C_VEL
LIN {X 0,Y 270.414,Z 462.677,A -85,B 0,C 180,E1 -18290.937,E2 -18290.937} C_VEL
LIN {X 0,Y 270.459,Z 465.779,A -85,B 0,C 180,E1 -18291.333,E2 -18291.333} C_VEL
LIN {X 0,Y 268.915,Z 477.083,A -85,B 0,C 180,E1 -18292.876,E2 -18292.876} C_VEL
LIN {X 0,Y 267.401,Z 486.757,A -85,B 0,C 180,E1 -18294.525,E2 -18294.525} C_VEL
LIN {X 0,Y 265.931,Z 495.545,A -85,B 0,C 180,E1 -18296.357,E2 -18296.357} C_VEL
LIN {X 0,Y 264.518,Z 504.152,A -85,B 0,C 180,E1 -18298.57,E2 -18298.57} C_VEL
LIN {X 0,Y 263.319,Z 511.281,A -85,B 0,C 180,E1 -18300.868,E2 -18300.868} C_VEL
LIN {X 0,Y 262.423,Z 516.764,A -85,B 0,C 180,E1 -18303.079,E2 -18303.079} C_VEL
LIN {X 0,Y 261.813,Z 521.043,A -85,B 0,C 180,E1 -18305.248,E2 -18305.248} C_VEL
LIN {X 0,Y 261.372,Z 524.085,A -85,B 0,C 180,E1 -18307.227,E2 -18307.227} C_VEL
LIN {X 0,Y 261.138,Z 525.875,A -85,B 0,C 180,E1 -18308.696,E2 -18308.696} C_VEL
LIN {X 0,Y 260.909,Z 527.91,A -85,B 0,C 180,E1 -18311.042,E2 -18311.042} C_VEL
LIN {X 0,Y 260.811,Z 528.971,A -85,B 0,C 180,E1 -18313.318,E2 -18313.318} C_VEL
LIN {X 0,Y 260.939,Z 529.169,A -85,B 0,C 180,E1 -18315.551,E2 -18315.551} C_VEL
LIN {X 0,Y 261.489,Z 527.988,A -85,B 0,C 180,E1 -18318.81,E2 -18318.81} C_VEL
LIN {X 0,Y 262.129,Z 526.164,A -85,B 0,C 180,E1 -18321.033,E2 -18321.033} C_VEL
LIN {X 0,Y 263.373,Z 522.216,A -85,B 0,C 180,E1 -18324.051,E2 -18324.051} C_VEL
LIN {X 0,Y 264.769,Z 517.58,A -85,B 0,C 180,E1 -18326.555,E2 -18326.555} C_VEL
LIN {X 0,Y 266.602,Z 511.443,A -85,B 0,C 180,E1 -18329.066,E2 -18329.066} C_VEL
LIN {X 0,Y 268.379,Z 505.3,A -85,B 0,C 180,E1 -18331.057,E2 -18331.057} C_VEL
LIN {X 0,Y 270.623,Z 497.353,A -85,B 0,C 180,E1 -18333.128,E2 -18333.128} C_VEL
LIN {X 0,Y 273.068,Z 487.824,A -85,B 0,C 180,E1 -18335.134,E2 -18335.134} C_VEL
LIN {X 0,Y 275.339,Z 478.163,A -85,B 0,C 180,E1 -18336.763,E2 -18336.763} C_VEL
LIN {X 0,Y 276.557,Z 471.04,A -85,B 0,C 180,E1 -18337.789,E2 -18337.789} C_VEL
LIN {X 0,Y 275.224,Z 461.429,A -85,B 0,C 180,E1 -18339.347,E2 -18339.347} C_VEL
LIN {X 0,Y 272.626,Z 450.625,A -85,B 0,C 180,E1 -18341.007,E2 -18341.007} C_VEL
LIN {X 0,Y 269.457,Z 441.113,A -85,B 0,C 180,E1 -18342.419,E2 -18342.419} C_VEL
LIN {X 0,Y 264.99,Z 430.725,A -85,B 0,C 180,E1 -18343.955,E2 -18343.955} C_VEL
LIN {X 0,Y 263.683,Z 427.67,A -85,B 0,C 180,E1 -18344.386,E2 -18344.386} C_VEL
LIN {X 0,Y 263.555,Z 427.051,A -85,B 0,C 180,E1 -18344.472,E2 -18344.472} C_VEL
LIN {X 0,Y 263.922,Z 424.946,A -85,B 0,C 180,E1 -18347.7,E2 -18347.7} C_VEL
LIN {X 0,Y 264.222,Z 423.062,A -85,B 0,C 180,E1 -18350.817,E2 -18350.817} C_VEL
LIN {X 0,Y 264.085,Z 421.441,A -85,B 0,C 180,E1 -18353.889,E2 -18353.889} C_VEL
LIN {X 0,Y 264.003,Z 419.3,A -85,B 0,C 180,E1 -18358.475,E2 -18358.475} C_VEL
LIN {X 0,Y 263.83,Z 418.126,A -85,B 0,C 180,E1 -18361.527,E2 -18361.527} C_VEL
LIN {X 0,Y 263.563,Z 417.655,A -85,B 0,C 180,E1 -18363.057,E2 -18363.057} C_VEL
LIN {X 0,Y 263.569,Z 417.656,A -85,B 0,C 180,E1 -18367.662,E2 -18367.662} C_VEL
LIN {X 0,Y 263.37,Z 417.679,A -85,B 0,C 180,E1 -18370.766,E2 -18370.766} C_VEL
LIN {X 0,Y 263.348,Z 417.683,A -85,B 0,C 180,E1 -18375.478,E2 -18375.478} C_VEL
LIN {X 0,Y 263.244,Z 417.694,A -85,B 0,C 180,E1 -18378.626,E2 -18378.626} C_VEL
LIN {X 0,Y 262.632,Z 417.777,A -85,B 0,C 180,E1 -18379.902,E2 -18379.902} C_VEL
LIN {X 0,Y 259.816,Z 418.129,A -85,B 0,C 180,E1 -18381.981,E2 -18381.981} C_VEL
LIN {X 0,Y 257.366,Z 418.429,A -85,B 0,C 180,E1 -18383.671,E2 -18383.671} C_VEL
LIN {X 0,Y 256.272,Z 418.562,A -85,B 0,C 180,E1 -18384.982,E2 -18384.982} C_VEL
LIN {X 0,Y 256.162,Z 418.575,A -85,B 0,C 180,E1 -18385.427,E2 -18385.427} C_VEL
LIN {X 0,Y 256.274,Z 419.289,A -85,B 0,C 180,E1 -18388.653,E2 -18388.653} C_VEL
LIN {X 0,Y 256.439,Z 420.51,A -85,B 0,C 180,E1 -18391.835,E2 -18391.835} C_VEL
LIN {X 0,Y 256.706,Z 422.035,A -85,B 0,C 180,E1 -18395.095,E2 -18395.095} C_VEL
LIN {X 0,Y 257.1,Z 424.215,A -85,B 0,C 180,E1 -18398.956,E2 -18398.956} C_VEL
LIN {X 0,Y 257.56,Z 426.936,A -85,B 0,C 180,E1 -18403.014,E2 -18403.014} C_VEL
LIN {X 0,Y 258.089,Z 430.295,A -85,B 0,C 180,E1 -18407.327,E2 -18407.327} C_VEL
LIN {X 0,Y 258.369,Z 432.287,A -85,B 0,C 180,E1 -18409.609,E2 -18409.609} C_VEL
LIN {X 0,Y 258.534,Z 434.531,A -85,B 0,C 180,E1 -18412.031,E2 -18412.031} C_VEL
LIN {X 0,Y 258.217,Z 437.717,A -85,B 0,C 180,E1 -18415.142,E2 -18415.142} C_VEL
LIN {X 0,Y 257.616,Z 440.354,A -85,B 0,C 180,E1 -18417.435,E2 -18417.435} C_VEL
LIN {X 0,Y 258.64,Z 443.786,A -85,B 0,C 180,E1 -18417.83,E2 -18417.83} C_VEL
LIN {X 0,Y 260.97,Z 450.391,A -85,B 0,C 180,E1 -18418.718,E2 -18418.718} C_VEL
LIN {X 0,Y 264.192,Z 461.379,A -85,B 0,C 180,E1 -18420.211,E2 -18420.211} C_VEL
LIN {X 0,Y 266.388,Z 473.124,A -85,B 0,C 180,E1 -18421.838,E2 -18421.838} C_VEL
LIN {X 0,Y 267.336,Z 484.068,A -85,B 0,C 180,E1 -18423.455,E2 -18423.455} C_VEL
LIN {X 0,Y 267.344,Z 494.419,A -85,B 0,C 180,E1 -18425.128,E2 -18425.128} C_VEL
LIN {X 0,Y 266.566,Z 500.076,A -85,B 0,C 180,E1 -18426.087,E2 -18426.087} C_VEL
LIN {X 0,Y 263.656,Z 510.739,A -85,B 0,C 180,E1 -18428.089,E2 -18428.089} C_VEL
LIN {X 0,Y 261.317,Z 519.166,A -85,B 0,C 180,E1 -18430.077,E2 -18430.077} C_VEL
LIN {X 0,Y 259.371,Z 526.583,A -85,B 0,C 180,E1 -18432.253,E2 -18432.253} C_VEL
LIN {X 0,Y 257.788,Z 531.994,A -85,B 0,C 180,E1 -18434.18,E2 -18434.18} C_VEL
LIN {X 0,Y 256.18,Z 537.344,A -85,B 0,C 180,E1 -18436.516,E2 -18436.516} C_VEL
LIN {X 0,Y 255.155,Z 541.547,A -85,B 0,C 180,E1 -18438.884,E2 -18438.884} C_VEL
LIN {X 0,Y 254.659,Z 543.788,A -85,B 0,C 180,E1 -18440.469,E2 -18440.469} C_VEL
LIN {X 0,Y 254.064,Z 546.935,A -85,B 0,C 180,E1 -18443.648,E2 -18443.648} C_VEL
LIN {X 0,Y 253.974,Z 547.92,A -85,B 0,C 180,E1 -18445.239,E2 -18445.239} C_VEL
LIN {X 0,Y 254.002,Z 548.503,A -85,B 0,C 180,E1 -18446.828,E2 -18446.828} C_VEL
LIN {X 0,Y 254.078,Z 548.655,A -85,B 0,C 180,E1 -18448.416,E2 -18448.416} C_VEL
LIN {X 0,Y 254.104,Z 548.41,A -85,B 0,C 180,E1 -18450.001,E2 -18450.001} C_VEL
LIN {X 0,Y 254.088,Z 547.768,A -85,B 0,C 180,E1 -18451.586,E2 -18451.586} C_VEL
LIN {X 0,Y 254.052,Z 546.709,A -85,B 0,C 180,E1 -18453.172,E2 -18453.172} C_VEL
LIN {X 0,Y 254.025,Z 544.772,A -85,B 0,C 180,E1 -18455.126,E2 -18455.126} C_VEL
LIN {X 0,Y 254.317,Z 540.832,A -85,B 0,C 180,E1 -18457.943,E2 -18457.943} C_VEL
LIN {X 0,Y 254.799,Z 536.26,A -85,B 0,C 180,E1 -18460.329,E2 -18460.329} C_VEL
LIN {X 0,Y 255.735,Z 529.296,A -85,B 0,C 180,E1 -18463.105,E2 -18463.105} C_VEL
LIN {X 0,Y 257.012,Z 521.756,A -85,B 0,C 180,E1 -18465.463,E2 -18465.463} C_VEL
LIN {X 0,Y 258.352,Z 514.062,A -85,B 0,C 180,E1 -18467.412,E2 -18467.412} C_VEL
LIN {X 0,Y 259.89,Z 504.698,A -85,B 0,C 180,E1 -18469.346,E2 -18469.346} C_VEL
LIN {X 0,Y 261.535,Z 494.347,A -85,B 0,C 180,E1 -18471.065,E2 -18471.065} C_VEL
LIN {X 0,Y 261.93,Z 490.331,A -85,B 0,C 180,E1 -18471.65,E2 -18471.65} C_VEL
LIN {X 0,Y 261.113,Z 479.025,A -85,B 0,C 180,E1 -18473.177,E2 -18473.177} C_VEL
LIN {X 0,Y 259.916,Z 467.476,A -85,B 0,C 180,E1 -18474.461,E2 -18474.461} C_VEL
LIN {X 0,Y 257.973,Z 454.58,A -85,B 0,C 180,E1 -18475.619,E2 -18475.619} C_VEL
LIN {X 0,Y 255.738,Z 442.687,A -85,B 0,C 180,E1 -18476.442,E2 -18476.442} C_VEL
LIN {X 0,Y 256.595,Z 437.623,A -85,B 0,C 180,E1 -18480.445,E2 -18480.445} C_VEL
LIN {X 0,Y 257.614,Z 431.916,A -85,B 0,C 180,E1 -18485.071,E2 -18485.071} C_VEL
LIN {X 0,Y 257.762,Z 428.758,A -85,B 0,C 180,E1 -18487.749,E2 -18487.749} C_VEL
LIN {X 0,Y 257.317,Z 425.162,A -85,B 0,C 180,E1 -18490.958,E2 -18490.958} C_VEL
LIN {X 0,Y 256.454,Z 420.441,A -85,B 0,C 180,E1 -18495.44,E2 -18495.44} C_VEL
LIN {X 0,Y 256.124,Z 418.584,A -85,B 0,C 180,E1 -18497.322,E2 -18497.322} C_VEL
LIN {X 0,Y 256.073,Z 418.591,A -85,B 0,C 180,E1 -18500.858,E2 -18500.858} C_VEL
LIN {X 0,Y 256.131,Z 418.58,A -85,B 0,C 180,E1 -18502.867,E2 -18502.867} C_VEL
LIN {X 0,Y 256.07,Z 418.587,A -85,B 0,C 180,E1 -18506.707,E2 -18506.707} C_VEL
LIN {X 0,Y 256.116,Z 418.58,A -85,B 0,C 180,E1 -18510.4,E2 -18510.4} C_VEL
LIN {X 0,Y 256.19,Z 418.569,A -85,B 0,C 180,E1 -18514.862,E2 -18514.862} C_VEL
LIN {X 0,Y 256.169,Z 418.577,A -85,B 0,C 180,E1 -18519.105,E2 -18519.105} C_VEL
LIN {X 0,Y 256.302,Z 418.556,A -85,B 0,C 180,E1 -18524.085,E2 -18524.085} C_VEL
LIN {X 0,Y 256.312,Z 418.556,A -85,B 0,C 180,E1 -18528.934,E2 -18528.934} C_VEL
LIN {X 0,Y 256.542,Z 418.526,A -85,B 0,C 180,E1 -18532.127,E2 -18532.127} C_VEL
LIN {X 0,Y 256.715,Z 418.504,A -85,B 0,C 180,E1 -18538.431,E2 -18538.431} C_VEL
LIN {X 0,Y 256.715,Z 418.504,A -85,B 0,C 180,E1 -18541.569,E2 -18541.569} C_VEL
LIN {X 0,Y 256.542,Z 418.525,A -85,B 0,C 180,E1 -18547.873,E2 -18547.873} C_VEL
LIN {X 0,Y 256.311,Z 418.556,A -85,B 0,C 180,E1 -18551.066,E2 -18551.066} C_VEL
LIN {X 0,Y 256.301,Z 418.548,A -85,B 0,C 180,E1 -18555.915,E2 -18555.915} C_VEL
LIN {X 0,Y 256.168,Z 418.569,A -85,B 0,C 180,E1 -18560.895,E2 -18560.895} C_VEL
LIN {X 0,Y 256.19,Z 418.572,A -85,B 0,C 180,E1 -18565.139,E2 -18565.139} C_VEL
LIN {X 0,Y 256.116,Z 418.579,A -85,B 0,C 180,E1 -18569.599,E2 -18569.599} C_VEL
LIN {X 0,Y 256.069,Z 418.579,A -85,B 0,C 180,E1 -18573.293,E2 -18573.293} C_VEL
LIN {X 0,Y 256.116,Z 418.573,A -85,B 0,C 180,E1 -18577.271,E2 -18577.271} C_VEL
LIN {X 0,Y 256.056,Z 418.587,A -85,B 0,C 180,E1 -18581.203,E2 -18581.203} C_VEL
LIN {X 0,Y 256.042,Z 418.588,A -85,B 0,C 180,E1 -18585.534,E2 -18585.534} C_VEL
LIN {X 0,Y 256.058,Z 418.583,A -85,B 0,C 180,E1 -18588.797,E2 -18588.797} C_VEL
LIN {X 0,Y 256.146,Z 418.575,A -85,B 0,C 180,E1 -18592.87,E2 -18592.87} C_VEL
LIN {X 0,Y 256.087,Z 418.587,A -85,B 0,C 180,E1 -18596.71,E2 -18596.71} C_VEL
LIN {X 0,Y 256.136,Z 418.574,A -85,B 0,C 180,E1 -18601.406,E2 -18601.406} C_VEL
LIN {X 0,Y 256.17,Z 418.572,A -85,B 0,C 180,E1 -18605.699,E2 -18605.699} C_VEL
LIN {X 0,Y 256.171,Z 418.573,A -85,B 0,C 180,E1 -18609.105,E2 -18609.105} C_VEL
LIN {X 0,Y 256.302,Z 418.558,A -85,B 0,C 180,E1 -18614.085,E2 -18614.085} C_VEL
LIN {X 0,Y 256.312,Z 418.555,A -85,B 0,C 180,E1 -18618.934,E2 -18618.934} C_VEL
LIN {X 0,Y 256.543,Z 418.53,A -85,B 0,C 180,E1 -18622.127,E2 -18622.127} C_VEL
LIN {X 0,Y 256.715,Z 418.509,A -85,B 0,C 180,E1 -18628.431,E2 -18628.431} C_VEL
LIN {X 0,Y 256.714,Z 418.506,A -85,B 0,C 180,E1 -18631.568,E2 -18631.568} C_VEL
LIN {X 0,Y 256.357,Z 418.554,A -85,B 0,C 180,E1 -18636.295,E2 -18636.295} C_VEL
LIN {X 0,Y 255.905,Z 418.708,A -85,B 0,C 180,E1 -18639.344,E2 -18639.344} C_VEL
LIN {X 0,Y 255.55,Z 421.515,A -85,B 0,C 180,E1 -18642.709,E2 -18642.709} C_VEL
LIN {X 0,Y 255.154,Z 424.847,A -85,B 0,C 180,E1 -18646.604,E2 -18646.604} C_VEL
LIN {X 0,Y 258.962,Z 439.617,A -85,B 0,C 180,E1 -18647.827,E2 -18647.827} C_VEL
LIN {X 0,Y 261.458,Z 451.223,A -85,B 0,C 180,E1 -18649.021,E2 -18649.021} C_VEL
LIN {X 0,Y 263.425,Z 463.107,A -85,B 0,C 180,E1 -18650.497,E2 -18650.497} C_VEL
LIN {X 0,Y 263.662,Z 466.114,A -85,B 0,C 180,E1 -18650.905,E2 -18650.905} C_VEL
LIN {X 0,Y 262.091,Z 477.26,A -85,B 0,C 180,E1 -18652.464,E2 -18652.464} C_VEL
LIN {X 0,Y 260.383,Z 487.727,A -85,B 0,C 180,E1 -18654.305,E2 -18654.305} C_VEL
LIN {X 0,Y 258.79,Z 497.043,A -85,B 0,C 180,E1 -18656.339,E2 -18656.339} C_VEL
LIN {X 0,Y 257.344,Z 505.52,A -85,B 0,C 180,E1 -18658.653,E2 -18658.653} C_VEL
LIN {X 0,Y 256.183,Z 512.271,A -85,B 0,C 180,E1 -18660.955,E2 -18660.955} C_VEL
LIN {X 0,Y 255.212,Z 518.013,A -85,B 0,C 180,E1 -18663.418,E2 -18663.418} C_VEL
LIN {X 0,Y 254.548,Z 522.756,A -85,B 0,C 180,E1 -18666.073,E2 -18666.073} C_VEL
LIN {X 0,Y 254.232,Z 524.692,A -85,B 0,C 180,E1 -18667.456,E2 -18667.456} C_VEL
LIN {X 0,Y 253.927,Z 526.928,A -85,B 0,C 180,E1 -18669.536,E2 -18669.536} C_VEL
LIN {X 0,Y 253.796,Z 528.475,A -85,B 0,C 180,E1 -18671.65,E2 -18671.65} C_VEL
LIN {X 0,Y 253.732,Z 529.36,A -85,B 0,C 180,E1 -18673.932,E2 -18673.932} C_VEL
LIN {X 0,Y 253.92,Z 529.422,A -85,B 0,C 180,E1 -18676.215,E2 -18676.215} C_VEL
LIN {X 0,Y 254.311,Z 528.657,A -85,B 0,C 180,E1 -18678.452,E2 -18678.452} C_VEL
LIN {X 0,Y 254.926,Z 527.141,A -85,B 0,C 180,E1 -18680.648,E2 -18680.648} C_VEL
LIN {X 0,Y 256.206,Z 523.473,A -85,B 0,C 180,E1 -18683.879,E2 -18683.879} C_VEL
LIN {X 0,Y 257.387,Z 519.86,A -85,B 0,C 180,E1 -18686.077,E2 -18686.077} C_VEL
LIN {X 0,Y 258.828,Z 515.247,A -85,B 0,C 180,E1 -18688.268,E2 -18688.268} C_VEL
LIN {X 0,Y 260.627,Z 509.563,A -85,B 0,C 180,E1 -18690.429,E2 -18690.429} C_VEL
LIN {X 0,Y 262.829,Z 502.513,A -85,B 0,C 180,E1 -18692.581,E2 -18692.581} C_VEL
LIN {X 0,Y 265.134,Z 494.462,A -85,B 0,C 180,E1 -18694.562,E2 -18694.562} C_VEL
LIN {X 0,Y 267.897,Z 483.772,A -85,B 0,C 180,E1 -18696.66,E2 -18696.66} C_VEL
LIN {X 0,Y 270.221,Z 473.59,A -85,B 0,C 180,E1 -18698.246,E2 -18698.246} C_VEL
LIN {X 0,Y 269.07,Z 463.646,A -85,B 0,C 180,E1 -18699.951,E2 -18699.951} C_VEL
LIN {X 0,Y 266.587,Z 452.689,A -85,B 0,C 180,E1 -18701.739,E2 -18701.739} C_VEL
LIN {X 0,Y 262.953,Z 441.982,A -85,B 0,C 180,E1 -18703.451,E2 -18703.451} C_VEL
LIN {X 0,Y 258.298,Z 431.301,A -85,B 0,C 180,E1 -18705.171,E2 -18705.171} C_VEL
LIN {X 0,Y 256.881,Z 428.385,A -85,B 0,C 180,E1 -18705.644,E2 -18705.644} C_VEL
LIN {X 0,Y 256.72,Z 427.41,A -85,B 0,C 180,E1 -18705.787,E2 -18705.787} C_VEL
LIN {X 0,Y 257.133,Z 425.026,A -85,B 0,C 180,E1 -18709.717,E2 -18709.717} C_VEL
LIN {X 0,Y 257.213,Z 423.702,A -85,B 0,C 180,E1 -18712.148,E2 -18712.148} C_VEL
LIN {X 0,Y 256.954,Z 422.198,A -85,B 0,C 180,E1 -18715.293,E2 -18715.293} C_VEL
LIN {X 0,Y 257.049,Z 420.787,A -85,B 0,C 180,E1 -18718.433,E2 -18718.433} C_VEL
LIN {X 0,Y 256.883,Z 419.64,A -85,B 0,C 180,E1 -18721.568,E2 -18721.568} C_VEL
LIN {X 0,Y 256.484,Z 418.538,A -85,B 0,C 180,E1 -18726.293,E2 -18726.293} C_VEL
LIN {X 0,Y 256.493,Z 418.535,A -85,B 0,C 180,E1 -18729.463,E2 -18729.463} C_VEL
LIN {X 0,Y 256.252,Z 418.566,A -85,B 0,C 180,E1 -18734.29,E2 -18734.29} C_VEL
LIN {X 0,Y 256.208,Z 418.571,A -85,B 0,C 180,E1 -18737.562,E2 -18737.562} C_VEL
LIN {X 0,Y 256.154,Z 418.577,A -85,B 0,C 180,E1 -18741.12,E2 -18741.12} C_VEL
LIN {X 0,Y 256.162,Z 418.575,A -85,B 0,C 180,E1 -18745.427,E2 -18745.427} C_VEL
LIN {X 0,Y 255.482,Z 418.894,A -85,B 0,C 180,E1 -18746.738,E2 -18746.738} C_VEL
LIN {X 0,Y 252.807,Z 420.22,A -85,B 0,C 180,E1 -18748.87,E2 -18748.87} C_VEL
LIN {X 0,Y 250.577,Z 421.42,A -85,B 0,C 180,E1 -18750.599,E2 -18750.599} C_VEL
LIN {X 0,Y 249.636,Z 422.202,A -85,B 0,C 180,E1 -18751.938,E2 -18751.938} C_VEL
LIN {X 0,Y 249.565,Z 422.419,A -85,B 0,C 180,E1 -18752.392,E2 -18752.392} C_VEL
LIN {X 0,Y 249.879,Z 424.242,A -85,B 0,C 180,E1 -18756.203,E2 -18756.203} C_VEL
LIN {X 0,Y 250.385,Z 426.874,A -85,B 0,C 180,E1 -18760.726,E2 -18760.726} C_VEL
LIN {X 0,Y 250.767,Z 429.487,A -85,B 0,C 180,E1 -18764.479,E2 -18764.479} C_VEL
LIN {X 0,Y 251.172,Z 432.1,A -85,B 0,C 180,E1 -18767.815,E2 -18767.815} C_VEL
LIN {X 0,Y 251.531,Z 435.289,A -85,B 0,C 180,E1 -18771.476,E2 -18771.476} C_VEL
LIN {X 0,Y 251.331,Z 437.93,A -85,B 0,C 180,E1 -18774.187,E2 -18774.187} C_VEL
LIN {X 0,Y 250.935,Z 439.915,A -85,B 0,C 180,E1 -18776.066,E2 -18776.066} C_VEL
LIN {X 0,Y 251.791,Z 442.958,A -85,B 0,C 180,E1 -18776.436,E2 -18776.436} C_VEL
LIN {X 0,Y 252.836,Z 445.538,A -85,B 0,C 180,E1 -18776.827,E2 -18776.827} C_VEL
LIN {X 0,Y 256.164,Z 455.484,A -85,B 0,C 180,E1 -18778.267,E2 -18778.267} C_VEL
LIN {X 0,Y 258.976,Z 466.917,A -85,B 0,C 180,E1 -18779.947,E2 -18779.947} C_VEL
LIN {X 0,Y 260.54,Z 477.152,A -85,B 0,C 180,E1 -18781.481,E2 -18781.481} C_VEL
LIN {X 0,Y 261.107,Z 488.592,A -85,B 0,C 180,E1 -18783.309,E2 -18783.309} C_VEL
LIN {X 0,Y 260.624,Z 498.613,A -85,B 0,C 180,E1 -18785.081,E2 -18785.081} C_VEL
LIN {X 0,Y 258.18,Z 507.724,A -85,B 0,C 180,E1 -18786.753,E2 -18786.753} C_VEL
LIN {X 0,Y 255.673,Z 516.142,A -85,B 0,C 180,E1 -18788.641,E2 -18788.641} C_VEL
LIN {X 0,Y 253.236,Z 524.412,A -85,B 0,C 180,E1 -18790.969,E2 -18790.969} C_VEL
LIN {X 0,Y 251.29,Z 531.144,A -85,B 0,C 180,E1 -18793.342,E2 -18793.342} C_VEL
LIN {X 0,Y 249.275,Z 537.401,A -85,B 0,C 180,E1 -18796.135,E2 -18796.135} C_VEL
LIN {X 0,Y 248.161,Z 541.521,A -85,B 0,C 180,E1 -18798.567,E2 -18798.567} C_VEL
LIN {X 0,Y 247.632,Z 543.691,A -85,B 0,C 180,E1 -18800.196,E2 -18800.196} C_VEL
LIN {X 0,Y 247.009,Z 546.773,A -85,B 0,C 180,E1 -18803.466,E2 -18803.466} C_VEL
LIN {X 0,Y 246.883,Z 547.723,A -85,B 0,C 180,E1 -18805.102,E2 -18805.102} C_VEL
LIN {X 0,Y 246.9,Z 548.242,A -85,B 0,C 180,E1 -18806.737,E2 -18806.737} C_VEL
LIN {X 0,Y 247.004,Z 548.361,A -85,B 0,C 180,E1 -18808.37,E2 -18808.37} C_VEL
LIN {X 0,Y 247.032,Z 548.086,A -85,B 0,C 180,E1 -18810.001,E2 -18810.001} C_VEL
LIN {X 0,Y 247.016,Z 547.414,A -85,B 0,C 180,E1 -18811.631,E2 -18811.631} C_VEL
LIN {X 0,Y 246.966,Z 546.292,A -85,B 0,C 180,E1 -18813.263,E2 -18813.263} C_VEL
LIN {X 0,Y 246.952,Z 544.532,A -85,B 0,C 180,E1 -18815.082,E2 -18815.082} C_VEL
LIN {X 0,Y 247.265,Z 540.299,A -85,B 0,C 180,E1 -18818.171,E2 -18818.171} C_VEL
LIN {X 0,Y 247.783,Z 535.647,A -85,B 0,C 180,E1 -18820.625,E2 -18820.625} C_VEL
LIN {X 0,Y 248.787,Z 528.599,A -85,B 0,C 180,E1 -18823.477,E2 -18823.477} C_VEL
LIN {X 0,Y 250.118,Z 520.967,A -85,B 0,C 180,E1 -18825.901,E2 -18825.901} C_VEL
LIN {X 0,Y 251.47,Z 513.147,A -85,B 0,C 180,E1 -18827.905,E2 -18827.905} C_VEL
LIN {X 0,Y 253.289,Z 502.552,A -85,B 0,C 180,E1 -18830.083,E2 -18830.083} C_VEL
LIN {X 0,Y 255.011,Z 491.822,A -85,B 0,C 180,E1 -18831.843,E2 -18831.843} C_VEL
LIN {X 0,Y 254.32,Z 480.64,A -85,B 0,C 180,E1 -18833.436,E2 -18833.436} C_VEL
LIN {X 0,Y 253.008,Z 467.702,A -85,B 0,C 180,E1 -18834.941,E2 -18834.941} C_VEL
LIN {X 0,Y 251.046,Z 454.666,A -85,B 0,C 180,E1 -18836.157,E2 -18836.157} C_VEL
LIN {X 0,Y 248.771,Z 442.423,A -85,B 0,C 180,E1 -18837.044,E2 -18837.044} C_VEL
LIN {X 0,Y 249.683,Z 437.137,A -85,B 0,C 180,E1 -18841.382,E2 -18841.382} C_VEL
LIN {X 0,Y 250.369,Z 433.807,A -85,B 0,C 180,E1 -18844.154,E2 -18844.154} C_VEL
LIN {X 0,Y 250.729,Z 430.411,A -85,B 0,C 180,E1 -18847.06,E2 -18847.06} C_VEL
LIN {X 0,Y 250.463,Z 426.962,A -85,B 0,C 180,E1 -18850.195,E2 -18850.195} C_VEL
LIN {X 0,Y 249.57,Z 422.226,A -85,B 0,C 180,E1 -18854.75,E2 -18854.75} C_VEL
LIN {X 0,Y 249.066,Z 419.463,A -85,B 0,C 180,E1 -18857.647,E2 -18857.647} C_VEL
LIN {X 0,Y 249.045,Z 419.461,A -85,B 0,C 180,E1 -18862.2,E2 -18862.2} C_VEL
LIN {X 0,Y 249.045,Z 419.462,A -85,B 0,C 180,E1 -18865.639,E2 -18865.639} C_VEL
LIN {X 0,Y 249.054,Z 419.461,A -85,B 0,C 180,E1 -18869.473,E2 -18869.473} C_VEL
LIN {X 0,Y 249.075,Z 419.454,A -85,B 0,C 180,E1 -18873.162,E2 -18873.162} C_VEL
LIN {X 0,Y 249.081,Z 419.457,A -85,B 0,C 180,E1 -18876.733,E2 -18876.733} C_VEL
LIN {X 0,Y 249.112,Z 419.452,A -85,B 0,C 180,E1 -18880.212,E2 -18880.212} C_VEL
LIN {X 0,Y 249.244,Z 419.437,A -85,B 0,C 180,E1 -18883.622,E2 -18883.622} C_VEL
LIN {X 0,Y 249.255,Z 419.434,A -85,B 0,C 180,E1 -18888.617,E2 -18888.617} C_VEL
LIN {X 0,Y 249.483,Z 419.406,A -85,B 0,C 180,E1 -18891.903,E2 -18891.903} C_VEL
LIN {X 0,Y 249.436,Z 419.411,A -85,B 0,C 180,E1 -18896.769,E2 -18896.769} C_VEL
LIN {X 0,Y 249.723,Z 419.375,A -85,B 0,C 180,E1 -18900,E2 -18900} C_VEL
LIN {X 0,Y 249.436,Z 419.411,A -85,B 0,C 180,E1 -18903.23,E2 -18903.23} C_VEL
LIN {X 0,Y 249.483,Z 419.405,A -85,B 0,C 180,E1 -18908.097,E2 -18908.097} C_VEL
LIN {X 0,Y 249.255,Z 419.433,A -85,B 0,C 180,E1 -18911.383,E2 -18911.383} C_VEL
LIN {X 0,Y 249.244,Z 419.427,A -85,B 0,C 180,E1 -18916.378,E2 -18916.378} C_VEL
LIN {X 0,Y 249.089,Z 419.45,A -85,B 0,C 180,E1 -18921.518,E2 -18921.518} C_VEL
LIN {X 0,Y 249.133,Z 419.45,A -85,B 0,C 180,E1 -18925.482,E2 -18925.482} C_VEL
LIN {X 0,Y 249.085,Z 419.457,A -85,B 0,C 180,E1 -18928.993,E2 -18928.993} C_VEL
LIN {X 0,Y 249.032,Z 419.461,A -85,B 0,C 180,E1 -18932.426,E2 -18932.426} C_VEL
LIN {X 0,Y 249.031,Z 419.45,A -85,B 0,C 180,E1 -18936.345,E2 -18936.345} C_VEL
LIN {X 0,Y 249.007,Z 419.464,A -85,B 0,C 180,E1 -18940.478,E2 -18940.478} C_VEL
LIN {X 0,Y 248.987,Z 419.469,A -85,B 0,C 180,E1 -18944.883,E2 -18944.883} C_VEL
LIN {X 0,Y 249.011,Z 419.462,A -85,B 0,C 180,E1 -18947.361,E2 -18947.361} C_VEL
LIN {X 0,Y 249.04,Z 419.452,A -85,B 0,C 180,E1 -18951.621,E2 -18951.621} C_VEL
LIN {X 0,Y 249.063,Z 419.457,A -85,B 0,C 180,E1 -18955.642,E2 -18955.642} C_VEL
LIN {X 0,Y 249.052,Z 419.459,A -85,B 0,C 180,E1 -18959.473,E2 -18959.473} C_VEL
LIN {X 0,Y 249.074,Z 419.452,A -85,B 0,C 180,E1 -18963.162,E2 -18963.162} C_VEL
LIN {X 0,Y 249.083,Z 419.459,A -85,B 0,C 180,E1 -18966.733,E2 -18966.733} C_VEL
LIN {X 0,Y 249.114,Z 419.454,A -85,B 0,C 180,E1 -18970.211,E2 -18970.211} C_VEL
LIN {X 0,Y 249.244,Z 419.435,A -85,B 0,C 180,E1 -18973.622,E2 -18973.622} C_VEL
LIN {X 0,Y 249.255,Z 419.435,A -85,B 0,C 180,E1 -18978.616,E2 -18978.616} C_VEL
LIN {X 0,Y 249.487,Z 419.408,A -85,B 0,C 180,E1 -18981.902,E2 -18981.902} C_VEL
LIN {X 0,Y 249.437,Z 419.411,A -85,B 0,C 180,E1 -18986.769,E2 -18986.769} C_VEL
LIN {X 0,Y 249.729,Z 419.379,A -85,B 0,C 180,E1 -18989.999,E2 -18989.999} C_VEL
LIN {X 0,Y 249.424,Z 419.411,A -85,B 0,C 180,E1 -18993.23,E2 -18993.23} C_VEL
LIN {X 0,Y 249.288,Z 419.434,A -85,B 0,C 180,E1 -18996.474,E2 -18996.474} C_VEL
LIN {X 0,Y 248.876,Z 419.53,A -85,B 0,C 180,E1 -18999.252,E2 -18999.252} C_VEL
LIN {X 0,Y 248.442,Z 422.689,A -85,B 0,C 180,E1 -19003.079,E2 -19003.079} C_VEL
LIN {X 0,Y 248.167,Z 425.263,A -85,B 0,C 180,E1 -19006.025,E2 -19006.025} C_VEL
LIN {X 0,Y 251.58,Z 438.176,A -85,B 0,C 180,E1 -19007.108,E2 -19007.108} C_VEL
LIN {X 0,Y 254.146,Z 450.007,A -85,B 0,C 180,E1 -19008.333,E2 -19008.333} C_VEL
LIN {X 0,Y 256.297,Z 462.026,A -85,B 0,C 180,E1 -19009.836,E2 -19009.836} C_VEL
LIN {X 0,Y 256.8,Z 466.97,A -85,B 0,C 180,E1 -19010.526,E2 -19010.526} C_VEL
LIN {X 0,Y 255.232,Z 477.659,A -85,B 0,C 180,E1 -19012.074,E2 -19012.074} C_VEL
LIN {X 0,Y 253.568,Z 487.515,A -85,B 0,C 180,E1 -19013.845,E2 -19013.845} C_VEL
LIN {X 0,Y 251.799,Z 497.51,A -85,B 0,C 180,E1 -19016.077,E2 -19016.077} C_VEL
LIN {X 0,Y 250.283,Z 506.115,A -85,B 0,C 180,E1 -19018.512,E2 -19018.512} C_VEL
LIN {X 0,Y 248.92,Z 513.749,A -85,B 0,C 180,E1 -19021.251,E2 -19021.251} C_VEL
LIN {X 0,Y 248.073,Z 518.74,A -85,B 0,C 180,E1 -19023.534,E2 -19023.534} C_VEL
LIN {X 0,Y 247.545,Z 522.325,A -85,B 0,C 180,E1 -19025.59,E2 -19025.59} C_VEL
LIN {X 0,Y 247.165,Z 524.668,A -85,B 0,C 180,E1 -19027.235,E2 -19027.235} C_VEL
LIN {X 0,Y 246.8,Z 527.338,A -85,B 0,C 180,E1 -19029.748,E2 -19029.748} C_VEL
LIN {X 0,Y 246.677,Z 528.978,A -85,B 0,C 180,E1 -19032.204,E2 -19032.204} C_VEL
LIN {X 0,Y 246.723,Z 529.775,A -85,B 0,C 180,E1 -19035.407,E2 -19035.407} C_VEL
LIN {X 0,Y 247.065,Z 529.404,A -85,B 0,C 180,E1 -19037.695,E2 -19037.695} C_VEL
LIN {X 0,Y 247.61,Z 528.204,A -85,B 0,C 180,E1 -19040.026,E2 -19040.026} C_VEL
LIN {X 0,Y 248.434,Z 526.15,A -85,B 0,C 180,E1 -19042.38,E2 -19042.38} C_VEL
LIN {X 0,Y 249.547,Z 523.17,A -85,B 0,C 180,E1 -19044.757,E2 -19044.757} C_VEL
LIN {X 0,Y 250.941,Z 519.129,A -85,B 0,C 180,E1 -19047.159,E2 -19047.159} C_VEL
LIN {X 0,Y 253.119,Z 512.764,A -85,B 0,C 180,E1 -19050.015,E2 -19050.015} C_VEL
LIN {X 0,Y 255.615,Z 505.224,A -85,B 0,C 180,E1 -19052.579,E2 -19052.579} C_VEL
LIN {X 0,Y 258.069,Z 497.366,A -85,B 0,C 180,E1 -19054.691,E2 -19054.691} C_VEL
LIN {X 0,Y 260.707,Z 488.126,A -85,B 0,C 180,E1 -19056.695,E2 -19056.695} C_VEL
LIN {X 0,Y 263.257,Z 478.193,A -85,B 0,C 180,E1 -19058.424,E2 -19058.424} C_VEL
LIN {X 0,Y 263.896,Z 474.32,A -85,B 0,C 180,E1 -19059.043,E2 -19059.043} C_VEL
LIN {X 0,Y 262.692,Z 464.238,A -85,B 0,C 180,E1 -19060.869,E2 -19060.869} C_VEL
LIN {X 0,Y 260.188,Z 453.6,A -85,B 0,C 180,E1 -19062.715,E2 -19062.715} C_VEL
LIN {X 0,Y 256.661,Z 443.138,A -85,B 0,C 180,E1 -19064.515,E2 -19064.515} C_VEL
LIN {X 0,Y 253.122,Z 435.143,A -85,B 0,C 180,E1 -19065.926,E2 -19065.926} C_VEL
LIN {X 0,Y 251.543,Z 431.77,A -85,B 0,C 180,E1 -19066.519,E2 -19066.519} C_VEL
LIN {X 0,Y 250.066,Z 428.761,A -85,B 0,C 180,E1 -19067.058,E2 -19067.058} C_VEL
LIN {X 0,Y 249.899,Z 427.809,A -85,B 0,C 180,E1 -19067.205,E2 -19067.205} C_VEL
LIN {X 0,Y 250.237,Z 426.037,A -85,B 0,C 180,E1 -19070.299,E2 -19070.299} C_VEL
LIN {X 0,Y 250.207,Z 424.388,A -85,B 0,C 180,E1 -19073.549,E2 -19073.549} C_VEL
LIN {X 0,Y 250.119,Z 422.301,A -85,B 0,C 180,E1 -19078.39,E2 -19078.39} C_VEL
LIN {X 0,Y 250.131,Z 421.684,A -85,B 0,C 180,E1 -19080,E2 -19080} C_VEL
LIN {X 0,Y 249.692,Z 420.713,A -85,B 0,C 180,E1 -19083.227,E2 -19083.227} C_VEL
LIN {X 0,Y 249.502,Z 419.562,A -85,B 0,C 180,E1 -19088.097,E2 -19088.097} C_VEL
LIN {X 0,Y 249.25,Z 419.439,A -85,B 0,C 180,E1 -19091.384,E2 -19091.384} C_VEL
LIN {X 0,Y 249.239,Z 419.44,A -85,B 0,C 180,E1 -19096.378,E2 -19096.378} C_VEL
LIN {X 0,Y 249.084,Z 419.458,A -85,B 0,C 180,E1 -19101.519,E2 -19101.519} C_VEL
LIN {X 0,Y 249.224,Z 420.089,A -85,B 0,C 180,E1 -19105.529,E2 -19105.529} C_VEL
LIN {X 0,Y 249.383,Z 421.15,A -85,B 0,C 180,E1 -19109.119,E2 -19109.119} C_VEL
LIN {X 0,Y 249.565,Z 422.419,A -85,B 0,C 180,E1 -19112.392,E2 -19112.392} C_VEL
LIN {X 0,Y 248.979,Z 423.186,A -85,B 0,C 180,E1 -19113.73,E2 -19113.73} C_VEL
LIN {X 0,Y 246.417,Z 424.898,A -85,B 0,C 180,E1 -19115.907,E2 -19115.907} C_VEL
LIN {X 0,Y 243.547,Z 427.064,A -85,B 0,C 180,E1 -19118.581,E2 -19118.581} C_VEL
LIN {X 0,Y 243.298,Z 427.683,A -85,B 0,C 180,E1 -19119.504,E2 -19119.504} C_VEL
LIN {X 0,Y 243.768,Z 430.538,A -85,B 0,C 180,E1 -19123.883,E2 -19123.883} C_VEL
LIN {X 0,Y 244.04,Z 432.288,A -85,B 0,C 180,E1 -19126.279,E2 -19126.279} C_VEL
LIN {X 0,Y 244.291,Z 434.096,A -85,B 0,C 180,E1 -19128.573,E2 -19128.573} C_VEL
LIN {X 0,Y 244.495,Z 436.085,A -85,B 0,C 180,E1 -19130.906,E2 -19130.906} C_VEL
LIN {X 0,Y 244.381,Z 438.591,A -85,B 0,C 180,E1 -19133.633,E2 -19133.633} C_VEL
LIN {X 0,Y 244.214,Z 439.507,A -85,B 0,C 180,E1 -19134.543,E2 -19134.543} C_VEL
LIN {X 0,Y 245.054,Z 442.541,A -85,B 0,C 180,E1 -19134.933,E2 -19134.933} C_VEL
LIN {X 0,Y 246.243,Z 444.91,A -85,B 0,C 180,E1 -19135.376,E2 -19135.376} C_VEL
LIN {X 0,Y 249.994,Z 456.114,A -85,B 0,C 180,E1 -19137.149,E2 -19137.149} C_VEL
LIN {X 0,Y 253.069,Z 468.978,A -85,B 0,C 180,E1 -19139.157,E2 -19139.157} C_VEL
LIN {X 0,Y 254.481,Z 479.773,A -85,B 0,C 180,E1 -19140.904,E2 -19140.904} C_VEL
LIN {X 0,Y 254.769,Z 491.43,A -85,B 0,C 180,E1 -19142.902,E2 -19142.902} C_VEL
LIN {X 0,Y 254.024,Z 500.517,A -85,B 0,C 180,E1 -19144.607,E2 -19144.607} C_VEL
LIN {X 0,Y 251.131,Z 510.094,A -85,B 0,C 180,E1 -19146.498,E2 -19146.498} C_VEL
LIN {X 0,Y 248.605,Z 518.032,A -85,B 0,C 180,E1 -19148.439,E2 -19148.439} C_VEL
LIN {X 0,Y 246.101,Z 526.066,A -85,B 0,C 180,E1 -19150.878,E2 -19150.878} C_VEL
LIN {X 0,Y 244.162,Z 532.324,A -85,B 0,C 180,E1 -19153.272,E2 -19153.272} C_VEL
LIN {X 0,Y 242.358,Z 537.466,A -85,B 0,C 180,E1 -19155.731,E2 -19155.731} C_VEL
LIN {X 0,Y 241.185,Z 541.505,A -85,B 0,C 180,E1 -19158.231,E2 -19158.231} C_VEL
LIN {X 0,Y 240.208,Z 545.307,A -85,B 0,C 180,E1 -19161.589,E2 -19161.589} C_VEL
LIN {X 0,Y 239.926,Z 546.611,A -85,B 0,C 180,E1 -19163.272,E2 -19163.272} C_VEL
LIN {X 0,Y 239.798,Z 547.585,A -85,B 0,C 180,E1 -19165.189,E2 -19165.189} C_VEL
LIN {X 0,Y 239.909,Z 548.068,A -85,B 0,C 180,E1 -19168.322,E2 -19168.322} C_VEL
LIN {X 0,Y 239.961,Z 547.76,A -85,B 0,C 180,E1 -19170.001,E2 -19170.001} C_VEL
LIN {X 0,Y 239.945,Z 547.04,A -85,B 0,C 180,E1 -19171.679,E2 -19171.679} C_VEL
LIN {X 0,Y 239.864,Z 545.861,A -85,B 0,C 180,E1 -19173.36,E2 -19173.36} C_VEL
LIN {X 0,Y 239.9,Z 543.31,A -85,B 0,C 180,E1 -19175.886,E2 -19175.886} C_VEL
LIN {X 0,Y 240.208,Z 539.717,A -85,B 0,C 180,E1 -19178.413,E2 -19178.413} C_VEL
LIN {X 0,Y 240.783,Z 534.982,A -85,B 0,C 180,E1 -19180.937,E2 -19180.937} C_VEL
LIN {X 0,Y 241.863,Z 527.843,A -85,B 0,C 180,E1 -19183.871,E2 -19183.871} C_VEL
LIN {X 0,Y 243.258,Z 520.064,A -85,B 0,C 180,E1 -19186.362,E2 -19186.362} C_VEL
LIN {X 0,Y 244.639,Z 512.102,A -85,B 0,C 180,E1 -19188.422,E2 -19188.422} C_VEL
LIN {X 0,Y 246.392,Z 502.431,A -85,B 0,C 180,E1 -19190.452,E2 -19190.452} C_VEL
LIN {X 0,Y 248.041,Z 493.035,A -85,B 0,C 180,E1 -19192.051,E2 -19192.051} C_VEL
LIN {X 0,Y 247.639,Z 484.164,A -85,B 0,C 180,E1 -19193.411,E2 -19193.411} C_VEL
LIN {X 0,Y 246.547,Z 471.845,A -85,B 0,C 180,E1 -19195.005,E2 -19195.005} C_VEL
LIN {X 0,Y 244.815,Z 458.991,A -85,B 0,C 180,E1 -19196.343,E2 -19196.343} C_VEL
LIN {X 0,Y 242.376,Z 445.457,A -85,B 0,C 180,E1 -19197.456,E2 -19197.456} C_VEL
LIN {X 0,Y 241.81,Z 442.145,A -85,B 0,C 180,E1 -19197.712,E2 -19197.712} C_VEL
LIN {X 0,Y 242.606,Z 437.736,A -85,B 0,C 180,E1 -19201.429,E2 -19201.429} C_VEL
LIN {X 0,Y 243.482,Z 433.287,A -85,B 0,C 180,E1 -19205.261,E2 -19205.261} C_VEL
LIN {X 0,Y 243.67,Z 431.038,A -85,B 0,C 180,E1 -19207.279,E2 -19207.279} C_VEL
LIN {X 0,Y 243.515,Z 428.715,A -85,B 0,C 180,E1 -19209.415,E2 -19209.415} C_VEL
LIN {X 0,Y 242.738,Z 424.413,A -85,B 0,C 180,E1 -19213.628,E2 -19213.628} C_VEL
LIN {X 0,Y 242.026,Z 420.341,A -85,B 0,C 180,E1 -19217.956,E2 -19217.956} C_VEL
LIN {X 0,Y 241.988,Z 420.34,A -85,B 0,C 180,E1 -19222.418,E2 -19222.418} C_VEL
LIN {X 0,Y 241.982,Z 420.341,A -85,B 0,C 180,E1 -19226.507,E2 -19226.507} C_VEL
LIN {X 0,Y 242.039,Z 420.334,A -85,B 0,C 180,E1 -19230.587,E2 -19230.587} C_VEL
LIN {X 0,Y 242.07,Z 420.325,A -85,B 0,C 180,E1 -19234.183,E2 -19234.183} C_VEL
LIN {X 0,Y 242.055,Z 420.332,A -85,B 0,C 180,E1 -19238.297,E2 -19238.297} C_VEL
LIN {X 0,Y 242.165,Z 420.32,A -85,B 0,C 180,E1 -19243.278,E2 -19243.278} C_VEL
LIN {X 0,Y 242.189,Z 420.312,A -85,B 0,C 180,E1 -19248.28,E2 -19248.28} C_VEL
LIN {X 0,Y 242.43,Z 420.285,A -85,B 0,C 180,E1 -19251.666,E2 -19251.666} C_VEL
LIN {X 0,Y 242.261,Z 420.306,A -85,B 0,C 180,E1 -19255.007,E2 -19255.007} C_VEL
LIN {X 0,Y 242.637,Z 420.257,A -85,B 0,C 180,E1 -19258.34,E2 -19258.34} C_VEL
LIN {X 0,Y 242.638,Z 420.258,A -85,B 0,C 180,E1 -19261.66,E2 -19261.66} C_VEL
LIN {X 0,Y 242.431,Z 420.283,A -85,B 0,C 180,E1 -19266.72,E2 -19266.72} C_VEL
LIN {X 0,Y 242.316,Z 420.298,A -85,B 0,C 180,E1 -19270.022,E2 -19270.022} C_VEL
LIN {X 0,Y 242.168,Z 420.309,A -85,B 0,C 180,E1 -19275.141,E2 -19275.141} C_VEL
LIN {X 0,Y 242.075,Z 420.314,A -85,B 0,C 180,E1 -19278.624,E2 -19278.624} C_VEL
LIN {X 0,Y 242.015,Z 420.331,A -85,B 0,C 180,E1 -19282.18,E2 -19282.18} C_VEL
LIN {X 0,Y 242.068,Z 420.329,A -85,B 0,C 180,E1 -19285.838,E2 -19285.838} C_VEL
LIN {X 0,Y 242.032,Z 420.333,A -85,B 0,C 180,E1 -19289.58,E2 -19289.58} C_VEL
LIN {X 0,Y 241.982,Z 420.331,A -85,B 0,C 180,E1 -19293.492,E2 -19293.492} C_VEL
LIN {X 0,Y 241.988,Z 420.33,A -85,B 0,C 180,E1 -19297.582,E2 -19297.582} C_VEL
LIN {X 0,Y 241.935,Z 420.345,A -85,B 0,C 180,E1 -19301.923,E2 -19301.923} C_VEL
LIN {X 0,Y 241.926,Z 420.349,A -85,B 0,C 180,E1 -19306.573,E2 -19306.573} C_VEL
LIN {X 0,Y 241.974,Z 420.335,A -85,B 0,C 180,E1 -19310.284,E2 -19310.284} C_VEL
LIN {X 0,Y 242.038,Z 420.333,A -85,B 0,C 180,E1 -19314.497,E2 -19314.497} C_VEL
LIN {X 0,Y 241.978,Z 420.345,A -85,B 0,C 180,E1 -19318.48,E2 -19318.48} C_VEL
LIN {X 0,Y 242.008,Z 420.335,A -85,B 0,C 180,E1 -19322.312,E2 -19322.312} C_VEL
LIN {X 0,Y 242.06,Z 420.331,A -85,B 0,C 180,E1 -19326.016,E2 -19326.016} C_VEL
LIN {X 0,Y 242.041,Z 420.333,A -85,B 0,C 180,E1 -19329.608,E2 -19329.608} C_VEL
LIN {X 0,Y 242.165,Z 420.317,A -85,B 0,C 180,E1 -19333.278,E2 -19333.278} C_VEL
LIN {X 0,Y 242.189,Z 420.317,A -85,B 0,C 180,E1 -19338.279,E2 -19338.279} C_VEL
LIN {X 0,Y 242.437,Z 420.285,A -85,B 0,C 180,E1 -19341.665,E2 -19341.665} C_VEL
LIN {X 0,Y 242.261,Z 420.301,A -85,B 0,C 180,E1 -19345.007,E2 -19345.007} C_VEL
LIN {X 0,Y 242.637,Z 420.261,A -85,B 0,C 180,E1 -19348.34,E2 -19348.34} C_VEL
LIN {X 0,Y 242.635,Z 420.261,A -85,B 0,C 180,E1 -19351.659,E2 -19351.659} C_VEL
LIN {X 0,Y 242.203,Z 420.315,A -85,B 0,C 180,E1 -19356.665,E2 -19356.665} C_VEL
LIN {X 0,Y 241.833,Z 420.423,A -85,B 0,C 180,E1 -19359.243,E2 -19359.243} C_VEL
LIN {X 0,Y 241.335,Z 423.828,A -85,B 0,C 180,E1 -19363.471,E2 -19363.471} C_VEL
LIN {X 0,Y 241.208,Z 425.387,A -85,B 0,C 180,E1 -19365.373,E2 -19365.373} C_VEL
LIN {X 0,Y 244.622,Z 438.494,A -85,B 0,C 180,E1 -19366.519,E2 -19366.519} C_VEL
LIN {X 0,Y 247.479,Z 451.766,A -85,B 0,C 180,E1 -19367.961,E2 -19367.961} C_VEL
LIN {X 0,Y 249.431,Z 463.032,A -85,B 0,C 180,E1 -19369.443,E2 -19369.443} C_VEL
LIN {X 0,Y 249.9,Z 467.895,A -85,B 0,C 180,E1 -19370.151,E2 -19370.151} C_VEL
LIN {X 0,Y 248.244,Z 478.85,A -85,B 0,C 180,E1 -19371.812,E2 -19371.812} C_VEL
LIN {X 0,Y 246.467,Z 489.164,A -85,B 0,C 180,E1 -19373.76,E2 -19373.76} C_VEL
LIN {X 0,Y 244.739,Z 498.477,A -85,B 0,C 180,E1 -19375.947,E2 -19375.947} C_VEL
LIN {X 0,Y 243.165,Z 507.031,A -85,B 0,C 180,E1 -19378.481,E2 -19378.481} C_VEL
LIN {X 0,Y 241.886,Z 513.926,A -85,B 0,C 180,E1 -19381.044,E2 -19381.044} C_VEL
LIN {X 0,Y 240.922,Z 519.454,A -85,B 0,C 180,E1 -19383.658,E2 -19383.658} C_VEL
LIN {X 0,Y 240.395,Z 522.956,A -85,B 0,C 180,E1 -19385.781,E2 -19385.781} C_VEL
LIN {X 0,Y 239.942,Z 525.776,A -85,B 0,C 180,E1 -19387.958,E2 -19387.958} C_VEL
LIN {X 0,Y 239.674,Z 528.013,A -85,B 0,C 180,E1 -19390.323,E2 -19390.323} C_VEL
LIN {X 0,Y 239.559,Z 529.483,A -85,B 0,C 180,E1 -19392.825,E2 -19392.825} C_VEL
LIN {X 0,Y 239.612,Z 530.046,A -85,B 0,C 180,E1 -19395.256,E2 -19395.256} C_VEL
LIN {X 0,Y 239.956,Z 529.78,A -85,B 0,C 180,E1 -19397.651,E2 -19397.651} C_VEL
LIN {X 0,Y 240.498,Z 528.762,A -85,B 0,C 180,E1 -19399.992,E2 -19399.992} C_VEL
LIN {X 0,Y 241.295,Z 527.012,A -85,B 0,C 180,E1 -19402.291,E2 -19402.291} C_VEL
LIN {X 0,Y 242.918,Z 522.937,A -85,B 0,C 180,E1 -19405.656,E2 -19405.656} C_VEL
LIN {X 0,Y 244.665,Z 518.219,A -85,B 0,C 180,E1 -19408.388,E2 -19408.388} C_VEL
LIN {X 0,Y 246.904,Z 512.077,A -85,B 0,C 180,E1 -19411.06,E2 -19411.06} C_VEL
LIN {X 0,Y 249.639,Z 504.264,A -85,B 0,C 180,E1 -19413.688,E2 -19413.688} C_VEL
LIN {X 0,Y 252.365,Z 495.966,A -85,B 0,C 180,E1 -19415.894,E2 -19415.894} C_VEL
LIN {X 0,Y 255.08,Z 486.716,A -85,B 0,C 180,E1 -19417.856,E2 -19417.856} C_VEL
LIN {X 0,Y 257.601,Z 477.164,A -85,B 0,C 180,E1 -19419.488,E2 -19419.488} C_VEL
LIN {X 0,Y 256.969,Z 469.076,A -85,B 0,C 180,E1 -19421.048,E2 -19421.048} C_VEL
LIN {X 0,Y 255.041,Z 458.771,A -85,B 0,C 180,E1 -19422.975,E2 -19422.975} C_VEL
LIN {X 0,Y 251.976,Z 448.712,A -85,B 0,C 180,E1 -19424.842,E2 -19424.842} C_VEL
LIN {X 0,Y 248.171,Z 439.217,A -85,B 0,C 180,E1 -19426.645,E2 -19426.645} C_VEL
LIN {X 0,Y 246.686,Z 436.063,A -85,B 0,C 180,E1 -19427.257,E2 -19427.257} C_VEL
LIN {X 0,Y 244.902,Z 432.385,A -85,B 0,C 180,E1 -19427.968,E2 -19427.968} C_VEL
LIN {X 0,Y 243.314,Z 429.331,A -85,B 0,C 180,E1 -19428.579,E2 -19428.579} C_VEL
LIN {X 0,Y 243.073,Z 428.223,A -85,B 0,C 180,E1 -19428.762,E2 -19428.762} C_VEL
LIN {X 0,Y 243.254,Z 426.686,A -85,B 0,C 180,E1 -19431.694,E2 -19431.694} C_VEL
LIN {X 0,Y 243.08,Z 425.18,A -85,B 0,C 180,E1 -19435.024,E2 -19435.024} C_VEL
LIN {X 0,Y 243.176,Z 423.817,A -85,B 0,C 180,E1 -19438.344,E2 -19438.344} C_VEL
LIN {X 0,Y 243.196,Z 423.202,A -85,B 0,C 180,E1 -19440,E2 -19440} C_VEL
LIN {X 0,Y 242.753,Z 422.26,A -85,B 0,C 180,E1 -19443.32,E2 -19443.32} C_VEL
LIN {X 0,Y 242.57,Z 421.155,A -85,B 0,C 180,E1 -19448.33,E2 -19448.33} C_VEL
LIN {X 0,Y 242.273,Z 420.77,A -85,B 0,C 180,E1 -19451.716,E2 -19451.716} C_VEL
LIN {X 0,Y 242.211,Z 420.611,A -85,B 0,C 180,E1 -19456.762,E2 -19456.762} C_VEL
LIN {X 0,Y 242.161,Z 421.079,A -85,B 0,C 180,E1 -19461.769,E2 -19461.769} C_VEL
LIN {X 0,Y 242.331,Z 421.918,A -85,B 0,C 180,E1 -19465.969,E2 -19465.969} C_VEL
LIN {X 0,Y 242.506,Z 423.014,A -85,B 0,C 180,E1 -19469.61,E2 -19469.61} C_VEL
LIN {X 0,Y 242.708,Z 424.513,A -85,B 0,C 180,E1 -19473.379,E2 -19473.379} C_VEL
LIN {X 0,Y 243.061,Z 426.481,A -85,B 0,C 180,E1 -19477.388,E2 -19477.388} C_VEL
LIN {X 0,Y 243.298,Z 427.683,A -85,B 0,C 180,E1 -19479.504,E2 -19479.504} C_VEL
LIN {X 0,Y 242.72,Z 428.683,A -85,B 0,C 180,E1 -19480.869,E2 -19480.869} C_VEL
LIN {X 0,Y 240.102,Z 430.752,A -85,B 0,C 180,E1 -19483.086,E2 -19483.086} C_VEL
LIN {X 0,Y 237.929,Z 432.5,A -85,B 0,C 180,E1 -19484.887,E2 -19484.887} C_VEL
LIN {X 0,Y 237.102,Z 433.713,A -85,B 0,C 180,E1 -19486.283,E2 -19486.283} C_VEL
LIN {X 0,Y 237.092,Z 434.077,A -85,B 0,C 180,E1 -19486.755,E2 -19486.755} C_VEL
LIN {X 0,Y 237.437,Z 436.883,A -85,B 0,C 180,E1 -19490.317,E2 -19490.317} C_VEL
LIN {X 0,Y 237.466,Z 439.14,A -85,B 0,C 180,E1 -19492.843,E2 -19492.843} C_VEL
LIN {X 0,Y 238.454,Z 442.296,A -85,B 0,C 180,E1 -19493.326,E2 -19493.326} C_VEL
LIN {X 0,Y 239.76,Z 444.96,A -85,B 0,C 180,E1 -19493.871,E2 -19493.871} C_VEL
LIN {X 0,Y 242.483,Z 452.131,A -85,B 0,C 180,E1 -19495.141,E2 -19495.141} C_VEL
LIN {X 0,Y 245.66,Z 463.544,A -85,B 0,C 180,E1 -19497.074,E2 -19497.074} C_VEL
LIN {X 0,Y 247.698,Z 474.905,A -85,B 0,C 180,E1 -19498.996,E2 -19498.996} C_VEL
LIN {X 0,Y 248.536,Z 484.886,A -85,B 0,C 180,E1 -19500.746,E2 -19500.746} C_VEL
LIN {X 0,Y 248.282,Z 495.626,A -85,B 0,C 180,E1 -19502.76,E2 -19502.76} C_VEL
LIN {X 0,Y 247.403,Z 502.372,A -85,B 0,C 180,E1 -19504.104,E2 -19504.104} C_VEL
LIN {X 0,Y 244.122,Z 512.395,A -85,B 0,C 180,E1 -19506.232,E2 -19506.232} C_VEL
LIN {X 0,Y 241.043,Z 521.521,A -85,B 0,C 180,E1 -19508.716,E2 -19508.716} C_VEL
LIN {X 0,Y 238.731,Z 528.457,A -85,B 0,C 180,E1 -19511.106,E2 -19511.106} C_VEL
LIN {X 0,Y 236.688,Z 534.296,A -85,B 0,C 180,E1 -19513.616,E2 -19513.616} C_VEL
LIN {X 0,Y 234.943,Z 538.972,A -85,B 0,C 180,E1 -19516.155,E2 -19516.155} C_VEL
LIN {X 0,Y 233.886,Z 542.574,A -85,B 0,C 180,E1 -19518.737,E2 -19518.737} C_VEL
LIN {X 0,Y 233.177,Z 545.199,A -85,B 0,C 180,E1 -19521.333,E2 -19521.333} C_VEL
LIN {X 0,Y 232.872,Z 546.459,A -85,B 0,C 180,E1 -19523.067,E2 -19523.067} C_VEL
LIN {X 0,Y 232.707,Z 547.721,A -85,B 0,C 180,E1 -19526.538,E2 -19526.538} C_VEL
LIN {X 0,Y 232.815,Z 547.773,A -85,B 0,C 180,E1 -19528.271,E2 -19528.271} C_VEL
LIN {X 0,Y 232.891,Z 547.434,A -85,B 0,C 180,E1 -19530.001,E2 -19530.001} C_VEL
LIN {X 0,Y 232.852,Z 546.647,A -85,B 0,C 180,E1 -19531.73,E2 -19531.73} C_VEL
LIN {X 0,Y 232.77,Z 544.121,A -85,B 0,C 180,E1 -19534.883,E2 -19534.883} C_VEL
LIN {X 0,Y 233.035,Z 540.485,A -85,B 0,C 180,E1 -19537.8,E2 -19537.8} C_VEL
LIN {X 0,Y 233.541,Z 536.065,A -85,B 0,C 180,E1 -19540.403,E2 -19540.403} C_VEL
LIN {X 0,Y 234.317,Z 530.414,A -85,B 0,C 180,E1 -19543.001,E2 -19543.001} C_VEL
LIN {X 0,Y 235.688,Z 523.342,A -85,B 0,C 180,E1 -19545.568,E2 -19545.568} C_VEL
LIN {X 0,Y 237.265,Z 514.685,A -85,B 0,C 180,E1 -19548.066,E2 -19548.066} C_VEL
LIN {X 0,Y 238.933,Z 505.624,A -85,B 0,C 180,E1 -19550.175,E2 -19550.175} C_VEL
LIN {X 0,Y 240.771,Z 495.486,A -85,B 0,C 180,E1 -19552.075,E2 -19552.075} C_VEL
LIN {X 0,Y 241.121,Z 491.598,A -85,B 0,C 180,E1 -19552.719,E2 -19552.719} C_VEL
LIN {X 0,Y 240.413,Z 480.406,A -85,B 0,C 180,E1 -19554.429,E2 -19554.429} C_VEL
LIN {X 0,Y 239.207,Z 468.321,A -85,B 0,C 180,E1 -19555.949,E2 -19555.949} C_VEL
LIN {X 0,Y 237.287,Z 454.959,A -85,B 0,C 180,E1 -19557.309,E2 -19557.309} C_VEL
LIN {X 0,Y 234.86,Z 441.917,A -85,B 0,C 180,E1 -19558.339,E2 -19558.339} C_VEL
LIN {X 0,Y 235.753,Z 437.228,A -85,B 0,C 180,E1 -19562.453,E2 -19562.453} C_VEL
LIN {X 0,Y 236.462,Z 433.888,A -85,B 0,C 180,E1 -19565.421,E2 -19565.421} C_VEL
LIN {X 0,Y 236.534,Z 430.465,A -85,B 0,C 180,E1 -19568.606,E2 -19568.606} C_VEL
LIN {X 0,Y 236.022,Z 427.133,A -85,B 0,C 180,E1 -19571.89,E2 -19571.89} C_VEL
LIN {X 0,Y 235.205,Z 422.623,A -85,B 0,C 180,E1 -19576.587,E2 -19576.587} C_VEL
LIN {X 0,Y 234.965,Z 421.22,A -85,B 0,C 180,E1 -19578.3,E2 -19578.3} C_VEL
LIN {X 0,Y 234.921,Z 421.227,A -85,B 0,C 180,E1 -19581.079,E2 -19581.079} C_VEL
LIN {X 0,Y 234.928,Z 421.22,A -85,B 0,C 180,E1 -19585.361,E2 -19585.361} C_VEL
LIN {X 0,Y 234.934,Z 421.22,A -85,B 0,C 180,E1 -19589.432,E2 -19589.432} C_VEL
LIN {X 0,Y 234.996,Z 421.206,A -85,B 0,C 180,E1 -19593.794,E2 -19593.794} C_VEL
LIN {X 0,Y 235.013,Z 421.212,A -85,B 0,C 180,E1 -19598.97,E2 -19598.97} C_VEL
LIN {X 0,Y 235.098,Z 421.2,A -85,B 0,C 180,E1 -19603.059,E2 -19603.059} C_VEL
LIN {X 0,Y 235.149,Z 421.189,A -85,B 0,C 180,E1 -19607.924,E2 -19607.924} C_VEL
LIN {X 0,Y 235.379,Z 421.164,A -85,B 0,C 180,E1 -19611.414,E2 -19611.414} C_VEL
LIN {X 0,Y 235.406,Z 421.162,A -85,B 0,C 180,E1 -19613.141,E2 -19613.141} C_VEL
LIN {X 0,Y 235.597,Z 421.134,A -85,B 0,C 180,E1 -19618.29,E2 -19618.29} C_VEL
LIN {X 0,Y 235.597,Z 421.134,A -85,B 0,C 180,E1 -19621.709,E2 -19621.709} C_VEL
LIN {X 0,Y 235.406,Z 421.16,A -85,B 0,C 180,E1 -19626.858,E2 -19626.858} C_VEL
LIN {X 0,Y 235.24,Z 421.18,A -85,B 0,C 180,E1 -19630.326,E2 -19630.326} C_VEL
LIN {X 0,Y 235.115,Z 421.184,A -85,B 0,C 180,E1 -19635.606,E2 -19635.606} C_VEL
LIN {X 0,Y 235.01,Z 421.197,A -85,B 0,C 180,E1 -19639.205,E2 -19639.205} C_VEL
LIN {X 0,Y 234.963,Z 421.214,A -85,B 0,C 180,E1 -19642.883,E2 -19642.883} C_VEL
LIN {X 0,Y 234.972,Z 421.217,A -85,B 0,C 180,E1 -19646.657,E2 -19646.657} C_VEL
LIN {X 0,Y 234.933,Z 421.22,A -85,B 0,C 180,E1 -19650.567,E2 -19650.567} C_VEL
LIN {X 0,Y 234.928,Z 421.207,A -85,B 0,C 180,E1 -19654.638,E2 -19654.638} C_VEL
LIN {X 0,Y 234.943,Z 421.214,A -85,B 0,C 180,E1 -19658.944,E2 -19658.944} C_VEL
LIN {X 0,Y 234.88,Z 421.225,A -85,B 0,C 180,E1 -19663.488,E2 -19663.488} C_VEL
LIN {X 0,Y 234.879,Z 421.227,A -85,B 0,C 180,E1 -19666.512,E2 -19666.512} C_VEL
LIN {X 0,Y 234.957,Z 421.206,A -85,B 0,C 180,E1 -19671.086,E2 -19671.086} C_VEL
LIN {X 0,Y 234.962,Z 421.214,A -85,B 0,C 180,E1 -19675.367,E2 -19675.367} C_VEL
LIN {X 0,Y 234.97,Z 421.215,A -85,B 0,C 180,E1 -19680.157,E2 -19680.157} C_VEL
LIN {X 0,Y 234.996,Z 421.205,A -85,B 0,C 180,E1 -19683.793,E2 -19683.793} C_VEL
LIN {X 0,Y 235.014,Z 421.209,A -85,B 0,C 180,E1 -19688.97,E2 -19688.97} C_VEL
LIN {X 0,Y 235.098,Z 421.198,A -85,B 0,C 180,E1 -19693.059,E2 -19693.059} C_VEL
LIN {X 0,Y 235.149,Z 421.193,A -85,B 0,C 180,E1 -19697.923,E2 -19697.923} C_VEL
LIN {X 0,Y 235.393,Z 421.162,A -85,B 0,C 180,E1 -19701.414,E2 -19701.414} C_VEL
LIN {X 0,Y 235.408,Z 421.159,A -85,B 0,C 180,E1 -19703.141,E2 -19703.141} C_VEL
LIN {X 0,Y 235.597,Z 421.137,A -85,B 0,C 180,E1 -19708.29,E2 -19708.29} C_VEL
LIN {X 0,Y 235.594,Z 421.138,A -85,B 0,C 180,E1 -19711.709,E2 -19711.709} C_VEL
LIN {X 0,Y 235.121,Z 421.197,A -85,B 0,C 180,E1 -19716.866,E2 -19716.866} C_VEL
LIN {X 0,Y 234.772,Z 421.361,A -85,B 0,C 180,E1 -19719.273,E2 -19719.273} C_VEL
LIN {X 0,Y 234.195,Z 425.321,A -85,B 0,C 180,E1 -19724.333,E2 -19724.333} C_VEL
LIN {X 0,Y 234.158,Z 425.635,A -85,B 0,C 180,E1 -19724.724,E2 -19724.724} C_VEL
LIN {X 0,Y 237.622,Z 438.751,A -85,B 0,C 180,E1 -19725.902,E2 -19725.902} C_VEL
LIN {X 0,Y 240.491,Z 451.861,A -85,B 0,C 180,E1 -19727.368,E2 -19727.368} C_VEL
LIN {X 0,Y 242.372,Z 462.587,A -85,B 0,C 180,E1 -19728.819,E2 -19728.819} C_VEL
LIN {X 0,Y 243.057,Z 468.019,A -85,B 0,C 180,E1 -19729.641,E2 -19729.641} C_VEL
LIN {X 0,Y 241.323,Z 479.606,A -85,B 0,C 180,E1 -19731.458,E2 -19731.458} C_VEL
LIN {X 0,Y 239.417,Z 490.239,A -85,B 0,C 180,E1 -19733.544,E2 -19733.544} C_VEL
LIN {X 0,Y 237.612,Z 499.618,A -85,B 0,C 180,E1 -19735.865,E2 -19735.865} C_VEL
LIN {X 0,Y 236.023,Z 507.961,A -85,B 0,C 180,E1 -19738.451,E2 -19738.451} C_VEL
LIN {X 0,Y 234.737,Z 514.738,A -85,B 0,C 180,E1 -19741.094,E2 -19741.094} C_VEL
LIN {X 0,Y 233.789,Z 520.123,A -85,B 0,C 180,E1 -19743.787,E2 -19743.787} C_VEL
LIN {X 0,Y 233.188,Z 523.989,A -85,B 0,C 180,E1 -19746.28,E2 -19746.28} C_VEL
LIN {X 0,Y 232.649,Z 527.417,A -85,B 0,C 180,E1 -19749.373,E2 -19749.373} C_VEL
LIN {X 0,Y 232.49,Z 529.12,A -85,B 0,C 180,E1 -19751.684,E2 -19751.684} C_VEL
LIN {X 0,Y 232.446,Z 530.092,A -85,B 0,C 180,E1 -19754.058,E2 -19754.058} C_VEL
LIN {X 0,Y 232.652,Z 530.314,A -85,B 0,C 180,E1 -19756.467,E2 -19756.467} C_VEL
LIN {X 0,Y 233.121,Z 529.778,A -85,B 0,C 180,E1 -19758.909,E2 -19758.909} C_VEL
LIN {X 0,Y 233.858,Z 528.434,A -85,B 0,C 180,E1 -19761.384,E2 -19761.384} C_VEL
LIN {X 0,Y 234.903,Z 526.198,A -85,B 0,C 180,E1 -19763.88,E2 -19763.88} C_VEL
LIN {X 0,Y 236.686,Z 521.928,A -85,B 0,C 180,E1 -19767.086,E2 -19767.086} C_VEL
LIN {X 0,Y 238.789,Z 516.593,A -85,B 0,C 180,E1 -19769.977,E2 -19769.977} C_VEL
LIN {X 0,Y 241.261,Z 510.171,A -85,B 0,C 180,E1 -19772.633,E2 -19772.633} C_VEL
LIN {X 0,Y 243.761,Z 503.41,A -85,B 0,C 180,E1 -19774.833,E2 -19774.833} C_VEL
LIN {X 0,Y 246.848,Z 494.342,A -85,B 0,C 180,E1 -19777.175,E2 -19777.175} C_VEL
LIN {X 0,Y 249.906,Z 484.223,A -85,B 0,C 180,E1 -19779.253,E2 -19779.253} C_VEL
LIN {X 0,Y 251.397,Z 478.788,A -85,B 0,C 180,E1 -19780.186,E2 -19780.186} C_VEL
LIN {X 0,Y 250.735,Z 469.748,A -85,B 0,C 180,E1 -19782.042,E2 -19782.042} C_VEL
LIN {X 0,Y 248.547,Z 458.856,A -85,B 0,C 180,E1 -19784.207,E2 -19784.207} C_VEL
LIN {X 0,Y 245.236,Z 448.28,A -85,B 0,C 180,E1 -19786.324,E2 -19786.324} C_VEL
LIN {X 0,Y 242.573,Z 441.568,A -85,B 0,C 180,E1 -19787.687,E2 -19787.687} C_VEL
LIN {X 0,Y 239.864,Z 436.187,A -85,B 0,C 180,E1 -19788.886,E2 -19788.886} C_VEL
LIN {X 0,Y 238.401,Z 433.066,A -85,B 0,C 180,E1 -19789.54,E2 -19789.54} C_VEL
LIN {X 0,Y 236.721,Z 430.254,A -85,B 0,C 180,E1 -19790.225,E2 -19790.225} C_VEL
LIN {X 0,Y 236.269,Z 428.661,A -85,B 0,C 180,E1 -19790.476,E2 -19790.476} C_VEL
LIN {X 0,Y 236.298,Z 427.405,A -85,B 0,C 180,E1 -19793.168,E2 -19793.168} C_VEL
LIN {X 0,Y 236.244,Z 425.33,A -85,B 0,C 180,E1 -19798.295,E2 -19798.295} C_VEL
LIN {X 0,Y 236.269,Z 424.729,A -85,B 0,C 180,E1 -19800,E2 -19800} C_VEL
